LIN {X 0,Y 442.361,Z 632.864,A -85,B 0,C 180,E1 20654.481,E2 20654.481} C_VEL
LIN {X 0,Y 442.378,Z 633.008,A -85,B 0,C 180,E1 20653.963,E2 20653.963} C_VEL
LIN {X 0,Y 443.347,Z 635.847,A -85,B 0,C 180,E1 20653.617,E2 20653.617} C_VEL
LIN {X 0,Y 449.92,Z 650.433,A -85,B 0,C 180,E1 20651.693,E2 20651.693} C_VEL
LIN {X 0,Y 457.492,Z 669.791,A -85,B 0,C 180,E1 20649.312,E2 20649.312} C_VEL
LIN {X 0,Y 464.291,Z 690.305,A -85,B 0,C 180,E1 20646.967,E2 20646.967} C_VEL
LIN {X 0,Y 466.418,Z 698.2,A -85,B 0,C 180,E1 20646.121,E2 20646.121} C_VEL
LIN {X 0,Y 463.345,Z 744.603,A -85,B 0,C 180,E1 20642.434,E2 20642.434} C_VEL
LIN {X 0,Y 460.284,Z 791.954,A -85,B 0,C 180,E1 20638.689,E2 20638.689} C_VEL
LIN {X 0,Y 457.632,Z 840.214,A -85,B 0,C 180,E1 20634.996,E2 20634.996} C_VEL
LIN {X 0,Y 456.966,Z 857.735,A -85,B 0,C 180,E1 20633.736,E2 20633.736} C_VEL
LIN {X 0,Y 457.546,Z 865.068,A -85,B 0,C 180,E1 20633.578,E2 20633.578} C_VEL
LIN {X 0,Y 454.351,Z 1025.223,A -85,B 0,C 180,E1 20631.032,E2 20631.032} C_VEL
LIN {X 0,Y 453.962,Z 1043.295,A -85,B 0,C 180,E1 20630.535,E2 20630.535} C_VEL
LIN {X 0,Y 453.251,Z 1059.664,A -85,B 0,C 180,E1 20629.858,E2 20629.858} C_VEL
LIN {X 0,Y 452.212,Z 1075.509,A -85,B 0,C 180,E1 20628.965,E2 20628.965} C_VEL
LIN {X 0,Y 450.872,Z 1091.243,A -85,B 0,C 180,E1 20627.819,E2 20627.819} C_VEL
LIN {X 0,Y 449.462,Z 1105.194,A -85,B 0,C 180,E1 20626.542,E2 20626.542} C_VEL
LIN {X 0,Y 447.963,Z 1118.231,A -85,B 0,C 180,E1 20625.07,E2 20625.07} C_VEL
LIN {X 0,Y 446.506,Z 1129.751,A -85,B 0,C 180,E1 20623.465,E2 20623.465} C_VEL
LIN {X 0,Y 445.09,Z 1140.448,A -85,B 0,C 180,E1 20621.628,E2 20621.628} C_VEL
LIN {X 0,Y 443.836,Z 1149.901,A -85,B 0,C 180,E1 20619.595,E2 20619.595} C_VEL
LIN {X 0,Y 442.873,Z 1157.352,A -85,B 0,C 180,E1 20617.523,E2 20617.523} C_VEL
LIN {X 0,Y 442.159,Z 1163.241,A -85,B 0,C 180,E1 20615.318,E2 20615.318} C_VEL
LIN {X 0,Y 441.708,Z 1167.308,A -85,B 0,C 180,E1 20613.113,E2 20613.113} C_VEL
LIN {X 0,Y 441.474,Z 1169.774,A -85,B 0,C 180,E1 20610.777,E2 20610.777} C_VEL
LIN {X 0,Y 441.429,Z 1170.363,A -85,B 0,C 180,E1 20608.441,E2 20608.441} C_VEL
LIN {X 0,Y 441.579,Z 1169.177,A -85,B 0,C 180,E1 20606.103,E2 20606.103} C_VEL
LIN {X 0,Y 441.927,Z 1166.376,A -85,B 0,C 180,E1 20603.894,E2 20603.894} C_VEL
LIN {X 0,Y 442.053,Z 1165.325,A -85,B 0,C 180,E1 20603.317,E2 20603.317} C_VEL
LIN {X 0,Y 441.321,Z 1163.494,A -85,B 0,C 180,E1 20602.344,E2 20602.344} C_VEL
LIN {X 0,Y 436.574,Z 1158.567,A -85,B 0,C 180,E1 20600.104,E2 20600.104} C_VEL
LIN {X 0,Y 435.691,Z 1155.543,A -85,B 0,C 180,E1 20599.088,E2 20599.088} C_VEL
LIN {X 0,Y 435.74,Z 1155.097,A -85,B 0,C 180,E1 20598.953,E2 20598.953} C_VEL
LIN {X 0,Y 436.956,Z 1146.938,A -85,B 0,C 180,E1 20596.905,E2 20596.905} C_VEL
LIN {X 0,Y 438.441,Z 1136.934,A -85,B 0,C 180,E1 20594.929,E2 20594.929} C_VEL
LIN {X 0,Y 439.985,Z 1126.234,A -85,B 0,C 180,E1 20593.223,E2 20593.223} C_VEL
LIN {X 0,Y 441.676,Z 1113.643,A -85,B 0,C 180,E1 20591.589,E2 20591.589} C_VEL
LIN {X 0,Y 443.34,Z 1099.655,A -85,B 0,C 180,E1 20590.134,E2 20590.134} C_VEL
LIN {X 0,Y 444.89,Z 1084.381,A -85,B 0,C 180,E1 20588.863,E2 20588.863} C_VEL
LIN {X 0,Y 446.207,Z 1068.28,A -85,B 0,C 180,E1 20587.814,E2 20587.814} C_VEL
LIN {X 0,Y 447.186,Z 1051.309,A -85,B 0,C 180,E1 20586.994,E2 20586.994} C_VEL
LIN {X 0,Y 447.792,Z 1033.412,A -85,B 0,C 180,E1 20586.391,E2 20586.391} C_VEL
LIN {X 0,Y 448.019,Z 1011.916,A -85,B 0,C 180,E1 20585.965,E2 20585.965} C_VEL
LIN {X 0,Y 451.206,Z 862.917,A -85,B 0,C 180,E1 20583.572,E2 20583.572} C_VEL
LIN {X 0,Y 450.631,Z 858.057,A -85,B 0,C 180,E1 20583.441,E2 20583.441} C_VEL
LIN {X 0,Y 453.107,Z 811.957,A -85,B 0,C 180,E1 20579.937,E2 20579.937} C_VEL
LIN {X 0,Y 456.239,Z 765.453,A -85,B 0,C 180,E1 20576.249,E2 20576.249} C_VEL
LIN {X 0,Y 459.516,Z 719.315,A -85,B 0,C 180,E1 20572.548,E2 20572.548} C_VEL
LIN {X 0,Y 460.586,Z 701.904,A -85,B 0,C 180,E1 20571.141,E2 20571.141} C_VEL
LIN {X 0,Y 454.384,Z 682.18,A -85,B 0,C 180,E1 20568.854,E2 20568.854} C_VEL
LIN {X 0,Y 452.123,Z 675.599,A -85,B 0,C 180,E1 20568.03,E2 20568.03} C_VEL
LIN {X 0,Y 453.874,Z 676.346,A -85,B 0,C 180,E1 20567.783,E2 20567.783} C_VEL
LIN {X 0,Y 456.65,Z 675.663,A -85,B 0,C 180,E1 20567.463,E2 20567.463} C_VEL
LIN {X 0,Y 457.757,Z 675.439,A -85,B 0,C 180,E1 20567.335,E2 20567.335} C_VEL
LIN {X 0,Y 475.007,Z 699.868,A -85,B 0,C 180,E1 20564.535,E2 20564.535} C_VEL
LIN {X 0,Y 489.761,Z 721.8,A -85,B 0,C 180,E1 20562.337,E2 20562.337} C_VEL
LIN {X 0,Y 471.768,Z 976.974,A -85,B 0,C 180,E1 20557.054,E2 20557.054} C_VEL
LIN {X 0,Y 469.932,Z 1000.353,A -85,B 0,C 180,E1 20556.346,E2 20556.346} C_VEL
LIN {X 0,Y 467.68,Z 1022.366,A -85,B 0,C 180,E1 20555.476,E2 20555.476} C_VEL
LIN {X 0,Y 465.047,Z 1043.255,A -85,B 0,C 180,E1 20554.435,E2 20554.435} C_VEL
LIN {X 0,Y 461.875,Z 1064.722,A -85,B 0,C 180,E1 20553.136,E2 20553.136} C_VEL
LIN {X 0,Y 458.629,Z 1084.634,A -85,B 0,C 180,E1 20551.697,E2 20551.697} C_VEL
LIN {X 0,Y 455.16,Z 1103.712,A -85,B 0,C 180,E1 20550.054,E2 20550.054} C_VEL
LIN {X 0,Y 451.494,Z 1122.574,A -85,B 0,C 180,E1 20548.146,E2 20548.146} C_VEL
LIN {X 0,Y 447.975,Z 1139.989,A -85,B 0,C 180,E1 20546.085,E2 20546.085} C_VEL
LIN {X 0,Y 444.684,Z 1155.904,A -85,B 0,C 180,E1 20543.875,E2 20543.875} C_VEL
LIN {X 0,Y 441.628,Z 1170.646,A -85,B 0,C 180,E1 20541.478,E2 20541.478} C_VEL
LIN {X 0,Y 439.042,Z 1183.69,A -85,B 0,C 180,E1 20539.007,E2 20539.007} C_VEL
LIN {X 0,Y 436.819,Z 1195.499,A -85,B 0,C 180,E1 20536.353,E2 20536.353} C_VEL
LIN {X 0,Y 435.035,Z 1205.998,A -85,B 0,C 180,E1 20533.53,E2 20533.53} C_VEL
LIN {X 0,Y 433.8,Z 1214.56,A -85,B 0,C 180,E1 20530.76,E2 20530.76} C_VEL
LIN {X 0,Y 432.983,Z 1221.42,A -85,B 0,C 180,E1 20527.964,E2 20527.964} C_VEL
LIN {X 0,Y 432.473,Z 1227.215,A -85,B 0,C 180,E1 20524.907,E2 20524.907} C_VEL
LIN {X 0,Y 432.262,Z 1231,A -85,B 0,C 180,E1 20522.121,E2 20522.121} C_VEL
LIN {X 0,Y 432.189,Z 1233.379,A -85,B 0,C 180,E1 20519.205,E2 20519.205} C_VEL
LIN {X 0,Y 432.208,Z 1234.345,A -85,B 0,C 180,E1 20516.419,E2 20516.419} C_VEL
LIN {X 0,Y 432.276,Z 1233.807,A -85,B 0,C 180,E1 20513.625,E2 20513.625} C_VEL
LIN {X 0,Y 432.492,Z 1231.87,A -85,B 0,C 180,E1 20510.687,E2 20510.687} C_VEL
LIN {X 0,Y 432.906,Z 1228.535,A -85,B 0,C 180,E1 20507.867,E2 20507.867} C_VEL
LIN {X 0,Y 433.692,Z 1223.483,A -85,B 0,C 180,E1 20504.899,E2 20504.899} C_VEL
LIN {X 0,Y 434.909,Z 1217.159,A -85,B 0,C 180,E1 20502.057,E2 20502.057} C_VEL
LIN {X 0,Y 436.66,Z 1209.045,A -85,B 0,C 180,E1 20499.211,E2 20499.211} C_VEL
LIN {X 0,Y 439.038,Z 1199.132,A -85,B 0,C 180,E1 20496.37,E2 20496.37} C_VEL
LIN {X 0,Y 441.963,Z 1187.801,A -85,B 0,C 180,E1 20493.677,E2 20493.677} C_VEL
LIN {X 0,Y 445.374,Z 1174.918,A -85,B 0,C 180,E1 20491.115,E2 20491.115} C_VEL
LIN {X 0,Y 449.088,Z 1160.665,A -85,B 0,C 180,E1 20488.75,E2 20488.75} C_VEL
LIN {X 0,Y 452.879,Z 1145.755,A -85,B 0,C 180,E1 20486.65,E2 20486.65} C_VEL
LIN {X 0,Y 456.84,Z 1129.478,A -85,B 0,C 180,E1 20484.702,E2 20484.702} C_VEL
LIN {X 0,Y 460.685,Z 1112.341,A -85,B 0,C 180,E1 20482.965,E2 20482.965} C_VEL
LIN {X 0,Y 464.478,Z 1093.552,A -85,B 0,C 180,E1 20481.37,E2 20481.37} C_VEL
LIN {X 0,Y 467.935,Z 1073.587,A -85,B 0,C 180,E1 20479.97,E2 20479.97} C_VEL
LIN {X 0,Y 471.001,Z 1052.378,A -85,B 0,C 180,E1 20478.764,E2 20478.764} C_VEL
LIN {X 0,Y 473.486,Z 1030.442,A -85,B 0,C 180,E1 20477.783,E2 20477.783} C_VEL
LIN {X 0,Y 475.36,Z 1007.879,A -85,B 0,C 180,E1 20477.012,E2 20477.012} C_VEL
LIN {X 0,Y 478.712,Z 978.56,A -85,B 0,C 180,E1 20476.153,E2 20476.153} C_VEL
LIN {X 0,Y 484.513,Z 946.475,A -85,B 0,C 180,E1 20475.242,E2 20475.242} C_VEL
LIN {X 0,Y 493.348,Z 909.949,A -85,B 0,C 180,E1 20474.196,E2 20474.196} C_VEL
LIN {X 0,Y 491.563,Z 920.862,A -85,B 0,C 180,E1 20472.901,E2 20472.901} C_VEL
LIN {X 0,Y 491.452,Z 927.421,A -85,B 0,C 180,E1 20472.156,E2 20472.156} C_VEL
LIN {X 0,Y 485.87,Z 946.673,A -85,B 0,C 180,E1 20472.006,E2 20472.006} C_VEL
LIN {X 0,Y 480.627,Z 965.886,A -85,B 0,C 180,E1 20471.62,E2 20471.62} C_VEL
LIN {X 0,Y 476.101,Z 984.154,A -85,B 0,C 180,E1 20471.02,E2 20471.02} C_VEL
LIN {X 0,Y 467.969,Z 1021.759,A -85,B 0,C 180,E1 20469.32,E2 20469.32} C_VEL
LIN {X 0,Y 461.485,Z 1054.214,A -85,B 0,C 180,E1 20467.585,E2 20467.585} C_VEL
LIN {X 0,Y 455.667,Z 1086.671,A -85,B 0,C 180,E1 20465.558,E2 20465.558} C_VEL
LIN {X 0,Y 450.935,Z 1115.987,A -85,B 0,C 180,E1 20463.438,E2 20463.438} C_VEL
LIN {X 0,Y 446.734,Z 1144.254,A -85,B 0,C 180,E1 20461.086,E2 20461.086} C_VEL
LIN {X 0,Y 443.422,Z 1168.395,A -85,B 0,C 180,E1 20458.78,E2 20458.78} C_VEL
LIN {X 0,Y 440.588,Z 1189.873,A -85,B 0,C 180,E1 20456.413,E2 20456.413} C_VEL
LIN {X 0,Y 438.235,Z 1209.061,A -85,B 0,C 180,E1 20453.964,E2 20453.964} C_VEL
LIN {X 0,Y 436.417,Z 1224.669,A -85,B 0,C 180,E1 20451.648,E2 20451.648} C_VEL
LIN {X 0,Y 434.936,Z 1238.794,A -85,B 0,C 180,E1 20449.194,E2 20449.194} C_VEL
LIN {X 0,Y 433.801,Z 1250.64,A -85,B 0,C 180,E1 20446.747,E2 20446.747} C_VEL
LIN {X 0,Y 433.012,Z 1260.497,A -85,B 0,C 180,E1 20444.306,E2 20444.306} C_VEL
LIN {X 0,Y 432.506,Z 1268.942,A -85,B 0,C 180,E1 20441.74,E2 20441.74} C_VEL
LIN {X 0,Y 432.226,Z 1275.553,A -85,B 0,C 180,E1 20439.187,E2 20439.187} C_VEL
LIN {X 0,Y 432.141,Z 1280.686,A -85,B 0,C 180,E1 20436.512,E2 20436.512} C_VEL
LIN {X 0,Y 432.145,Z 1283.861,A -85,B 0,C 180,E1 20433.982,E2 20433.982} C_VEL
LIN {X 0,Y 432.171,Z 1285.546,A -85,B 0,C 180,E1 20431.328,E2 20431.328} C_VEL
LIN {X 0,Y 432.169,Z 1285.595,A -85,B 0,C 180,E1 20428.676,E2 20428.676} C_VEL
LIN {X 0,Y 432.137,Z 1284.048,A -85,B 0,C 180,E1 20426.021,E2 20426.021} C_VEL
LIN {X 0,Y 432.118,Z 1280.876,A -85,B 0,C 180,E1 20423.358,E2 20423.358} C_VEL
LIN {X 0,Y 432.221,Z 1275.811,A -85,B 0,C 180,E1 20420.548,E2 20420.548} C_VEL
LIN {X 0,Y 432.552,Z 1268.98,A -85,B 0,C 180,E1 20417.723,E2 20417.723} C_VEL
LIN {X 0,Y 433.259,Z 1259.669,A -85,B 0,C 180,E1 20414.726,E2 20414.726} C_VEL
LIN {X 0,Y 434.381,Z 1248.907,A -85,B 0,C 180,E1 20411.898,E2 20411.898} C_VEL
LIN {X 0,Y 436.057,Z 1235.907,A -85,B 0,C 180,E1 20409.042,E2 20409.042} C_VEL
LIN {X 0,Y 438.251,Z 1221.293,A -85,B 0,C 180,E1 20406.327,E2 20406.327} C_VEL
LIN {X 0,Y 440.94,Z 1205.226,A -85,B 0,C 180,E1 20403.759,E2 20403.759} C_VEL
LIN {X 0,Y 444.345,Z 1186.33,A -85,B 0,C 180,E1 20401.163,E2 20401.163} C_VEL
LIN {X 0,Y 448.432,Z 1164.856,A -85,B 0,C 180,E1 20398.649,E2 20398.649} C_VEL
LIN {X 0,Y 452.655,Z 1143.094,A -85,B 0,C 180,E1 20396.482,E2 20396.482} C_VEL
LIN {X 0,Y 457.071,Z 1120.987,A -85,B 0,C 180,E1 20394.572,E2 20394.572} C_VEL
LIN {X 0,Y 461.561,Z 1097.922,A -85,B 0,C 180,E1 20392.887,E2 20392.887} C_VEL
LIN {X 0,Y 466.241,Z 1073.881,A -85,B 0,C 180,E1 20391.389,E2 20391.389} C_VEL
LIN {X 0,Y 470.405,Z 1051.347,A -85,B 0,C 180,E1 20390.226,E2 20390.226} C_VEL
LIN {X 0,Y 474.759,Z 1026.579,A -85,B 0,C 180,E1 20389.163,E2 20389.163} C_VEL
LIN {X 0,Y 478.579,Z 1001.615,A -85,B 0,C 180,E1 20388.317,E2 20388.317} C_VEL
LIN {X 0,Y 481.845,Z 975.438,A -85,B 0,C 180,E1 20387.621,E2 20387.621} C_VEL
LIN {X 0,Y 485.239,Z 953.953,A -85,B 0,C 180,E1 20387.28,E2 20387.28} C_VEL
LIN {X 0,Y 485.44,Z 951.656,A -85,B 0,C 180,E1 20387.232,E2 20387.232} C_VEL
LIN {X 0,Y 475.455,Z 930.968,A -85,B 0,C 180,E1 20385.71,E2 20385.71} C_VEL
LIN {X 0,Y 473.644,Z 926.121,A -85,B 0,C 180,E1 20385.351,E2 20385.351} C_VEL
LIN {X 0,Y 470.533,Z 906.683,A -85,B 0,C 180,E1 20383.011,E2 20383.011} C_VEL
LIN {X 0,Y 469.842,Z 885.654,A -85,B 0,C 180,E1 20380.633,E2 20380.633} C_VEL
LIN {X 0,Y 471.699,Z 862.2,A -85,B 0,C 180,E1 20378.15,E2 20378.15} C_VEL
LIN {X 0,Y 478.112,Z 821.82,A -85,B 0,C 180,E1 20374.089,E2 20374.089} C_VEL
LIN {X 0,Y 483.755,Z 787.898,A -85,B 0,C 180,E1 20370.638,E2 20370.638} C_VEL
LIN {X 0,Y 489.081,Z 756.617,A -85,B 0,C 180,E1 20367.387,E2 20367.387} C_VEL
LIN {X 0,Y 482.488,Z 739.607,A -85,B 0,C 180,E1 20364.356,E2 20364.356} C_VEL
LIN {X 0,Y 475.807,Z 723.064,A -85,B 0,C 180,E1 20361.189,E2 20361.189} C_VEL
LIN {X 0,Y 468.783,Z 706.507,A -85,B 0,C 180,E1 20357.759,E2 20357.759} C_VEL
LIN {X 0,Y 461.708,Z 690.572,A -85,B 0,C 180,E1 20354.165,E2 20354.165} C_VEL
LIN {X 0,Y 455.438,Z 677.174,A -85,B 0,C 180,E1 20350.883,E2 20350.883} C_VEL
LIN {X 0,Y 449.891,Z 665.361,A -85,B 0,C 180,E1 20347.792,E2 20347.792} C_VEL
LIN {X 0,Y 445.031,Z 655.663,A -85,B 0,C 180,E1 20345.027,E2 20345.027} C_VEL
LIN {X 0,Y 442.88,Z 651.358,A -85,B 0,C 180,E1 20343.75,E2 20343.75} C_VEL
LIN {X 0,Y 440.804,Z 647.144,A -85,B 0,C 180,E1 20342.47,E2 20342.47} C_VEL
LIN {X 0,Y 438.787,Z 642.92,A -85,B 0,C 180,E1 20341.175,E2 20341.175} C_VEL
LIN {X 0,Y 436.932,Z 639.254,A -85,B 0,C 180,E1 20339.98,E2 20339.98} C_VEL
LIN {X 0,Y 434.526,Z 634.515,A -85,B 0,C 180,E1 20338.418,E2 20338.418} C_VEL
LIN {X 0,Y 434.411,Z 633.857,A -85,B 0,C 180,E1 20338.153,E2 20338.153} C_VEL
LIN {X 0,Y 434.42,Z 633.869,A -85,B 0,C 180,E1 20334.32,E2 20334.32} C_VEL
LIN {X 0,Y 434.41,Z 633.863,A -85,B 0,C 180,E1 20330.594,E2 20330.594} C_VEL
LIN {X 0,Y 434.421,Z 633.855,A -85,B 0,C 180,E1 20326.693,E2 20326.693} C_VEL
LIN {X 0,Y 434.416,Z 633.857,A -85,B 0,C 180,E1 20323.003,E2 20323.003} C_VEL
LIN {X 0,Y 434.41,Z 633.861,A -85,B 0,C 180,E1 20319.239,E2 20319.239} C_VEL
LIN {X 0,Y 434.422,Z 633.863,A -85,B 0,C 180,E1 20315.38,E2 20315.38} C_VEL
LIN {X 0,Y 434.425,Z 633.863,A -85,B 0,C 180,E1 20311.544,E2 20311.544} C_VEL
LIN {X 0,Y 434.412,Z 633.866,A -85,B 0,C 180,E1 20307.724,E2 20307.724} C_VEL
LIN {X 0,Y 434.415,Z 633.859,A -85,B 0,C 180,E1 20304.06,E2 20304.06} C_VEL
LIN {X 0,Y 434.424,Z 633.863,A -85,B 0,C 180,E1 20300.219,E2 20300.219} C_VEL
LIN {X 0,Y 434.41,Z 633.817,A -85,B 0,C 180,E1 20296.329,E2 20296.329} C_VEL
LIN {X 0,Y 434.418,Z 633.853,A -85,B 0,C 180,E1 20294.771,E2 20294.771} C_VEL
LIN {X 0,Y 435.357,Z 636.731,A -85,B 0,C 180,E1 20294.416,E2 20294.416} C_VEL
LIN {X 0,Y 439.742,Z 646.024,A -85,B 0,C 180,E1 20293.122,E2 20293.122} C_VEL
LIN {X 0,Y 447.436,Z 664.476,A -85,B 0,C 180,E1 20290.73,E2 20290.73} C_VEL
LIN {X 0,Y 454.706,Z 684.886,A -85,B 0,C 180,E1 20288.275,E2 20288.275} C_VEL
LIN {X 0,Y 459.428,Z 700.781,A -85,B 0,C 180,E1 20286.5,E2 20286.5} C_VEL
LIN {X 0,Y 456.328,Z 745.479,A -85,B 0,C 180,E1 20282.913,E2 20282.913} C_VEL
LIN {X 0,Y 453.203,Z 792.434,A -85,B 0,C 180,E1 20279.18,E2 20279.18} C_VEL
LIN {X 0,Y 450.475,Z 840.077,A -85,B 0,C 180,E1 20275.504,E2 20275.504} C_VEL
LIN {X 0,Y 449.716,Z 858.67,A -85,B 0,C 180,E1 20274.153,E2 20274.153} C_VEL
LIN {X 0,Y 450.277,Z 866.044,A -85,B 0,C 180,E1 20273.992,E2 20273.992} C_VEL
LIN {X 0,Y 446.961,Z 1025.867,A -85,B 0,C 180,E1 20271.414,E2 20271.414} C_VEL
LIN {X 0,Y 446.556,Z 1044.024,A -85,B 0,C 180,E1 20270.909,E2 20270.909} C_VEL
LIN {X 0,Y 445.799,Z 1060.815,A -85,B 0,C 180,E1 20270.205,E2 20270.205} C_VEL
LIN {X 0,Y 444.719,Z 1076.607,A -85,B 0,C 180,E1 20269.298,E2 20269.298} C_VEL
LIN {X 0,Y 443.33,Z 1092.314,A -85,B 0,C 180,E1 20268.132,E2 20268.132} C_VEL
LIN {X 0,Y 441.843,Z 1106.464,A -85,B 0,C 180,E1 20266.813,E2 20266.813} C_VEL
LIN {X 0,Y 440.24,Z 1119.753,A -85,B 0,C 180,E1 20265.274,E2 20265.274} C_VEL
LIN {X 0,Y 438.68,Z 1131.583,A -85,B 0,C 180,E1 20263.576,E2 20263.576} C_VEL
LIN {X 0,Y 437.25,Z 1141.953,A -85,B 0,C 180,E1 20261.741,E2 20261.741} C_VEL
LIN {X 0,Y 436.009,Z 1150.899,A -85,B 0,C 180,E1 20259.769,E2 20259.769} C_VEL
LIN {X 0,Y 435,Z 1158.338,A -85,B 0,C 180,E1 20257.659,E2 20257.659} C_VEL
LIN {X 0,Y 434.252,Z 1164.219,A -85,B 0,C 180,E1 20255.415,E2 20255.415} C_VEL
LIN {X 0,Y 433.778,Z 1168.278,A -85,B 0,C 180,E1 20253.169,E2 20253.169} C_VEL
LIN {X 0,Y 433.533,Z 1170.732,A -85,B 0,C 180,E1 20250.791,E2 20250.791} C_VEL
LIN {X 0,Y 433.486,Z 1171.314,A -85,B 0,C 180,E1 20248.412,E2 20248.412} C_VEL
LIN {X 0,Y 433.647,Z 1170.121,A -85,B 0,C 180,E1 20246.032,E2 20246.032} C_VEL
LIN {X 0,Y 434.017,Z 1167.313,A -85,B 0,C 180,E1 20243.782,E2 20243.782} C_VEL
LIN {X 0,Y 434.642,Z 1162.71,A -85,B 0,C 180,E1 20241.532,E2 20241.532} C_VEL
LIN {X 0,Y 435.576,Z 1156.142,A -85,B 0,C 180,E1 20239.267,E2 20239.267} C_VEL
LIN {X 0,Y 435.74,Z 1155.097,A -85,B 0,C 180,E1 20238.953,E2 20238.953} C_VEL
LIN {X 0,Y 435.289,Z 1151.958,A -85,B 0,C 180,E1 20238.02,E2 20238.02} C_VEL
LIN {X 0,Y 431.73,Z 1145.302,A -85,B 0,C 180,E1 20236.204,E2 20236.204} C_VEL
LIN {X 0,Y 430.511,Z 1140.757,A -85,B 0,C 180,E1 20235.199,E2 20235.199} C_VEL
LIN {X 0,Y 430.603,Z 1138.835,A -85,B 0,C 180,E1 20234.836,E2 20234.836} C_VEL
LIN {X 0,Y 432.368,Z 1127.107,A -85,B 0,C 180,E1 20232.919,E2 20232.919} C_VEL
LIN {X 0,Y 434.13,Z 1114.495,A -85,B 0,C 180,E1 20231.257,E2 20231.257} C_VEL
LIN {X 0,Y 435.836,Z 1100.708,A -85,B 0,C 180,E1 20229.8,E2 20229.8} C_VEL
LIN {X 0,Y 437.397,Z 1085.929,A -85,B 0,C 180,E1 20228.544,E2 20228.544} C_VEL
LIN {X 0,Y 438.753,Z 1070.125,A -85,B 0,C 180,E1 20227.487,E2 20227.487} C_VEL
LIN {X 0,Y 439.79,Z 1053.487,A -85,B 0,C 180,E1 20226.651,E2 20226.651} C_VEL
LIN {X 0,Y 440.432,Z 1035.997,A -85,B 0,C 180,E1 20226.035,E2 20226.035} C_VEL
LIN {X 0,Y 440.682,Z 1016.129,A -85,B 0,C 180,E1 20225.61,E2 20225.61} C_VEL
LIN {X 0,Y 444.041,Z 863.864,A -85,B 0,C 180,E1 20223.126,E2 20223.126} C_VEL
LIN {X 0,Y 443.473,Z 859.061,A -85,B 0,C 180,E1 20222.995,E2 20222.995} C_VEL
LIN {X 0,Y 445.981,Z 814.116,A -85,B 0,C 180,E1 20219.555,E2 20219.555} C_VEL
LIN {X 0,Y 449.23,Z 767.039,A -85,B 0,C 180,E1 20215.804,E2 20215.804} C_VEL
LIN {X 0,Y 452.602,Z 721.3,A -85,B 0,C 180,E1 20212.108,E2 20212.108} C_VEL
LIN {X 0,Y 453.655,Z 704.806,A -85,B 0,C 180,E1 20210.758,E2 20210.758} C_VEL
LIN {X 0,Y 447.346,Z 684.549,A -85,B 0,C 180,E1 20208.341,E2 20208.341} C_VEL
LIN {X 0,Y 449.089,Z 685.28,A -85,B 0,C 180,E1 20208.09,E2 20208.09} C_VEL
LIN {X 0,Y 451.836,Z 684.583,A -85,B 0,C 180,E1 20207.763,E2 20207.763} C_VEL
LIN {X 0,Y 453.495,Z 684.211,A -85,B 0,C 180,E1 20207.569,E2 20207.569} C_VEL
LIN {X 0,Y 455.12,Z 684.122,A -85,B 0,C 180,E1 20207.372,E2 20207.372} C_VEL
LIN {X 0,Y 470.635,Z 706.14,A -85,B 0,C 180,E1 20204.839,E2 20204.839} C_VEL
LIN {X 0,Y 483.472,Z 725.409,A -85,B 0,C 180,E1 20202.882,E2 20202.882} C_VEL
LIN {X 0,Y 464.924,Z 977.284,A -85,B 0,C 180,E1 20197.559,E2 20197.559} C_VEL
LIN {X 0,Y 462.962,Z 1001.559,A -85,B 0,C 180,E1 20196.813,E2 20196.813} C_VEL
LIN {X 0,Y 460.532,Z 1024.321,A -85,B 0,C 180,E1 20195.889,E2 20195.889} C_VEL
LIN {X 0,Y 457.648,Z 1046.328,A -85,B 0,C 180,E1 20194.763,E2 20194.763} C_VEL
LIN {X 0,Y 454.42,Z 1067.268,A -85,B 0,C 180,E1 20193.449,E2 20193.449} C_VEL
LIN {X 0,Y 450.743,Z 1088.767,A -85,B 0,C 180,E1 20191.828,E2 20191.828} C_VEL
LIN {X 0,Y 447.189,Z 1107.79,A -85,B 0,C 180,E1 20190.131,E2 20190.131} C_VEL
LIN {X 0,Y 443.573,Z 1125.568,A -85,B 0,C 180,E1 20188.254,E2 20188.254} C_VEL
LIN {X 0,Y 439.805,Z 1143.593,A -85,B 0,C 180,E1 20186.026,E2 20186.026} C_VEL
LIN {X 0,Y 436.496,Z 1159.188,A -85,B 0,C 180,E1 20183.776,E2 20183.776} C_VEL
LIN {X 0,Y 433.492,Z 1173.353,A -85,B 0,C 180,E1 20181.373,E2 20181.373} C_VEL
LIN {X 0,Y 430.72,Z 1186.835,A -85,B 0,C 180,E1 20178.685,E2 20178.685} C_VEL
LIN {X 0,Y 428.554,Z 1198.321,A -85,B 0,C 180,E1 20175.981,E2 20175.981} C_VEL
LIN {X 0,Y 426.902,Z 1207.9,A -85,B 0,C 180,E1 20173.27,E2 20173.27} C_VEL
LIN {X 0,Y 425.64,Z 1216.58,A -85,B 0,C 180,E1 20170.285,E2 20170.285} C_VEL
LIN {X 0,Y 424.889,Z 1223.242,A -85,B 0,C 180,E1 20167.437,E2 20167.437} C_VEL
LIN {X 0,Y 424.452,Z 1228.23,A -85,B 0,C 180,E1 20164.594,E2 20164.594} C_VEL
LIN {X 0,Y 424.256,Z 1232.01,A -85,B 0,C 180,E1 20161.621,E2 20161.621} C_VEL
LIN {X 0,Y 424.204,Z 1234.09,A -85,B 0,C 180,E1 20158.784,E2 20158.784} C_VEL
LIN {X 0,Y 424.228,Z 1234.843,A -85,B 0,C 180,E1 20155.674,E2 20155.674} C_VEL
LIN {X 0,Y 424.359,Z 1234.079,A -85,B 0,C 180,E1 20152.745,E2 20152.745} C_VEL
LIN {X 0,Y 424.625,Z 1231.795,A -85,B 0,C 180,E1 20149.828,E2 20149.828} C_VEL
LIN {X 0,Y 425.204,Z 1227.975,A -85,B 0,C 180,E1 20146.795,E2 20146.795} C_VEL
LIN {X 0,Y 426.19,Z 1222.575,A -85,B 0,C 180,E1 20143.788,E2 20143.788} C_VEL
LIN {X 0,Y 427.739,Z 1215.379,A -85,B 0,C 180,E1 20140.755,E2 20140.755} C_VEL
LIN {X 0,Y 429.958,Z 1206.349,A -85,B 0,C 180,E1 20137.724,E2 20137.724} C_VEL
LIN {X 0,Y 432.665,Z 1196.259,A -85,B 0,C 180,E1 20134.949,E2 20134.949} C_VEL
LIN {X 0,Y 435.967,Z 1184.372,A -85,B 0,C 180,E1 20132.252,E2 20132.252} C_VEL
LIN {X 0,Y 439.559,Z 1171.576,A -85,B 0,C 180,E1 20129.817,E2 20129.817} C_VEL
LIN {X 0,Y 443.724,Z 1156.639,A -85,B 0,C 180,E1 20127.414,E2 20127.414} C_VEL
LIN {X 0,Y 447.913,Z 1141.065,A -85,B 0,C 180,E1 20125.302,E2 20125.302} C_VEL
LIN {X 0,Y 452.078,Z 1124.597,A -85,B 0,C 180,E1 20123.407,E2 20123.407} C_VEL
LIN {X 0,Y 456.398,Z 1105.826,A -85,B 0,C 180,E1 20121.603,E2 20121.603} C_VEL
LIN {X 0,Y 460.354,Z 1086.475,A -85,B 0,C 180,E1 20120.062,E2 20120.062} C_VEL
LIN {X 0,Y 463.78,Z 1066.993,A -85,B 0,C 180,E1 20118.777,E2 20118.777} C_VEL
LIN {X 0,Y 466.898,Z 1045.987,A -85,B 0,C 180,E1 20117.652,E2 20117.652} C_VEL
LIN {X 0,Y 469.446,Z 1024.223,A -85,B 0,C 180,E1 20116.733,E2 20116.733} C_VEL
LIN {X 0,Y 472.881,Z 994.654,A -85,B 0,C 180,E1 20115.751,E2 20115.751} C_VEL
LIN {X 0,Y 478.194,Z 966.7,A -85,B 0,C 180,E1 20114.891,E2 20114.891} C_VEL
LIN {X 0,Y 486.634,Z 934.282,A -85,B 0,C 180,E1 20113.931,E2 20113.931} C_VEL
LIN {X 0,Y 489.317,Z 925.284,A -85,B 0,C 180,E1 20113.649,E2 20113.649} C_VEL
LIN {X 0,Y 488.556,Z 930.278,A -85,B 0,C 180,E1 20113.053,E2 20113.053} C_VEL
LIN {X 0,Y 482.971,Z 949.556,A -85,B 0,C 180,E1 20112.878,E2 20112.878} C_VEL
LIN {X 0,Y 477.573,Z 968.489,A -85,B 0,C 180,E1 20112.472,E2 20112.472} C_VEL
LIN {X 0,Y 472.734,Z 986.225,A -85,B 0,C 180,E1 20111.862,E2 20111.862} C_VEL
LIN {X 0,Y 463.443,Z 1023.785,A -85,B 0,C 180,E1 20110.094,E2 20110.094} C_VEL
LIN {X 0,Y 456.064,Z 1056.427,A -85,B 0,C 180,E1 20108.271,E2 20108.271} C_VEL
LIN {X 0,Y 449.291,Z 1090.143,A -85,B 0,C 180,E1 20106.062,E2 20106.062} C_VEL
LIN {X 0,Y 443.848,Z 1120.553,A -85,B 0,C 180,E1 20103.741,E2 20103.741} C_VEL
LIN {X 0,Y 439.027,Z 1150.054,A -85,B 0,C 180,E1 20101.132,E2 20101.132} C_VEL
LIN {X 0,Y 435.44,Z 1174.145,A -85,B 0,C 180,E1 20098.682,E2 20098.682} C_VEL
LIN {X 0,Y 432.481,Z 1195.161,A -85,B 0,C 180,E1 20096.207,E2 20096.207} C_VEL
LIN {X 0,Y 430.083,Z 1213.424,A -85,B 0,C 180,E1 20093.718,E2 20093.718} C_VEL
LIN {X 0,Y 428.165,Z 1229.129,A -85,B 0,C 180,E1 20091.223,E2 20091.223} C_VEL
LIN {X 0,Y 426.696,Z 1242.474,A -85,B 0,C 180,E1 20088.727,E2 20088.727} C_VEL
LIN {X 0,Y 425.619,Z 1253.67,A -85,B 0,C 180,E1 20086.236,E2 20086.236} C_VEL
LIN {X 0,Y 424.842,Z 1263.46,A -85,B 0,C 180,E1 20083.585,E2 20083.585} C_VEL
LIN {X 0,Y 424.386,Z 1271.478,A -85,B 0,C 180,E1 20080.866,E2 20080.866} C_VEL
LIN {X 0,Y 424.181,Z 1277.626,A -85,B 0,C 180,E1 20078.133,E2 20078.133} C_VEL
LIN {X 0,Y 424.143,Z 1281.751,A -85,B 0,C 180,E1 20075.548,E2 20075.548} C_VEL
LIN {X 0,Y 424.17,Z 1284.335,A -85,B 0,C 180,E1 20072.839,E2 20072.839} C_VEL
LIN {X 0,Y 424.202,Z 1285.246,A -85,B 0,C 180,E1 20070.137,E2 20070.137} C_VEL
LIN {X 0,Y 424.171,Z 1284.523,A -85,B 0,C 180,E1 20067.435,E2 20067.435} C_VEL
LIN {X 0,Y 424.145,Z 1282.193,A -85,B 0,C 180,E1 20064.727,E2 20064.727} C_VEL
LIN {X 0,Y 424.165,Z 1277.956,A -85,B 0,C 180,E1 20061.871,E2 20061.871} C_VEL
LIN {X 0,Y 424.371,Z 1271.96,A -85,B 0,C 180,E1 20059,E2 20059} C_VEL
LIN {X 0,Y 424.835,Z 1264.508,A -85,B 0,C 180,E1 20056.251,E2 20056.251} C_VEL
LIN {X 0,Y 425.726,Z 1254.78,A -85,B 0,C 180,E1 20053.351,E2 20053.351} C_VEL
LIN {X 0,Y 427.062,Z 1243.588,A -85,B 0,C 180,E1 20050.584,E2 20050.584} C_VEL
LIN {X 0,Y 429.04,Z 1229.649,A -85,B 0,C 180,E1 20047.676,E2 20047.676} C_VEL
LIN {X 0,Y 431.573,Z 1214.037,A -85,B 0,C 180,E1 20044.916,E2 20044.916} C_VEL
LIN {X 0,Y 434.629,Z 1196.884,A -85,B 0,C 180,E1 20042.311,E2 20042.311} C_VEL
LIN {X 0,Y 438.417,Z 1177.142,A -85,B 0,C 180,E1 20039.736,E2 20039.736} C_VEL
LIN {X 0,Y 442.695,Z 1155.617,A -85,B 0,C 180,E1 20037.332,E2 20037.332} C_VEL
LIN {X 0,Y 447.58,Z 1131.425,A -85,B 0,C 180,E1 20035.042,E2 20035.042} C_VEL
LIN {X 0,Y 451.931,Z 1110.129,A -85,B 0,C 180,E1 20033.321,E2 20033.321} C_VEL
LIN {X 0,Y 456.996,Z 1084.983,A -85,B 0,C 180,E1 20031.586,E2 20031.586} C_VEL
LIN {X 0,Y 461.453,Z 1062.22,A -85,B 0,C 180,E1 20030.27,E2 20030.27} C_VEL
LIN {X 0,Y 466.29,Z 1036.214,A -85,B 0,C 180,E1 20029.035,E2 20029.035} C_VEL
LIN {X 0,Y 470.607,Z 1011.13,A -85,B 0,C 180,E1 20028.074,E2 20028.074} C_VEL
LIN {X 0,Y 474.137,Z 985.021,A -85,B 0,C 180,E1 20027.285,E2 20027.285} C_VEL
LIN {X 0,Y 476.92,Z 965.187,A -85,B 0,C 180,E1 20026.861,E2 20026.861} C_VEL
LIN {X 0,Y 478.68,Z 954.162,A -85,B 0,C 180,E1 20026.694,E2 20026.694} C_VEL
LIN {X 0,Y 469.464,Z 934.685,A -85,B 0,C 180,E1 20025.238,E2 20025.238} C_VEL
LIN {X 0,Y 465.374,Z 923.825,A -85,B 0,C 180,E1 20024.462,E2 20024.462} C_VEL
LIN {X 0,Y 462.989,Z 904.169,A -85,B 0,C 180,E1 20022.111,E2 20022.111} C_VEL
LIN {X 0,Y 463.032,Z 882.287,A -85,B 0,C 180,E1 20019.644,E2 20019.644} C_VEL
LIN {X 0,Y 465.656,Z 858.172,A -85,B 0,C 180,E1 20017.113,E2 20017.113} C_VEL
LIN {X 0,Y 471.492,Z 823.054,A -85,B 0,C 180,E1 20013.551,E2 20013.551} C_VEL
LIN {X 0,Y 477.402,Z 788.954,A -85,B 0,C 180,E1 20010.038,E2 20010.038} C_VEL
LIN {X 0,Y 482.411,Z 760.261,A -85,B 0,C 180,E1 20007.029,E2 20007.029} C_VEL
LIN {X 0,Y 475.302,Z 741.849,A -85,B 0,C 180,E1 20003.691,E2 20003.691} C_VEL
LIN {X 0,Y 468.163,Z 724.265,A -85,B 0,C 180,E1 20000.243,E2 20000.243} C_VEL
LIN {X 0,Y 460.923,Z 707.32,A -85,B 0,C 180,E1 19996.64,E2 19996.64} C_VEL
LIN {X 0,Y 454.108,Z 692.108,A -85,B 0,C 180,E1 19993.108,E2 19993.108} C_VEL
LIN {X 0,Y 447.945,Z 678.865,A -85,B 0,C 180,E1 19989.767,E2 19989.767} C_VEL
LIN {X 0,Y 442.006,Z 666.375,A -85,B 0,C 180,E1 19986.364,E2 19986.364} C_VEL
LIN {X 0,Y 437.216,Z 656.814,A -85,B 0,C 180,E1 19983.54,E2 19983.54} C_VEL
LIN {X 0,Y 435.084,Z 652.559,A -85,B 0,C 180,E1 19982.239,E2 19982.239} C_VEL
LIN {X 0,Y 432.983,Z 648.255,A -85,B 0,C 180,E1 19980.881,E2 19980.881} C_VEL
LIN {X 0,Y 430.567,Z 643.531,A -85,B 0,C 180,E1 19979.335,E2 19979.335} C_VEL
LIN {X 0,Y 428.418,Z 639.162,A -85,B 0,C 180,E1 19977.86,E2 19977.86} C_VEL
LIN {X 0,Y 426.646,Z 635.8,A -85,B 0,C 180,E1 19976.686,E2 19976.686} C_VEL
LIN {X 0,Y 426.474,Z 634.85,A -85,B 0,C 180,E1 19976.371,E2 19976.371} C_VEL
LIN {X 0,Y 426.487,Z 634.844,A -85,B 0,C 180,E1 19972.456,E2 19972.456} C_VEL
LIN {X 0,Y 426.471,Z 634.856,A -85,B 0,C 180,E1 19968.505,E2 19968.505} C_VEL
LIN {X 0,Y 426.486,Z 634.856,A -85,B 0,C 180,E1 19964.637,E2 19964.637} C_VEL
LIN {X 0,Y 426.484,Z 634.849,A -85,B 0,C 180,E1 19960.696,E2 19960.696} C_VEL
LIN {X 0,Y 426.472,Z 634.847,A -85,B 0,C 180,E1 19956.949,E2 19956.949} C_VEL
LIN {X 0,Y 426.476,Z 634.843,A -85,B 0,C 180,E1 19953.246,E2 19953.246} C_VEL
LIN {X 0,Y 426.483,Z 634.842,A -85,B 0,C 180,E1 19949.419,E2 19949.419} C_VEL
LIN {X 0,Y 426.481,Z 634.841,A -85,B 0,C 180,E1 19945.596,E2 19945.596} C_VEL
LIN {X 0,Y 426.475,Z 634.844,A -85,B 0,C 180,E1 19941.756,E2 19941.756} C_VEL
LIN {X 0,Y 426.475,Z 634.821,A -85,B 0,C 180,E1 19938.003,E2 19938.003} C_VEL
LIN {X 0,Y 426.495,Z 634.974,A -85,B 0,C 180,E1 19935.588,E2 19935.588} C_VEL
LIN {X 0,Y 427.888,Z 638.468,A -85,B 0,C 180,E1 19935.112,E2 19935.112} C_VEL
LIN {X 0,Y 435.286,Z 654.729,A -85,B 0,C 180,E1 19932.836,E2 19932.836} C_VEL
LIN {X 0,Y 442.672,Z 673.219,A -85,B 0,C 180,E1 19930.429,E2 19930.429} C_VEL
LIN {X 0,Y 449.641,Z 693.771,A -85,B 0,C 180,E1 19927.981,E2 19927.981} C_VEL
LIN {X 0,Y 452.428,Z 703.626,A -85,B 0,C 180,E1 19926.866,E2 19926.866} C_VEL
LIN {X 0,Y 449.186,Z 749.091,A -85,B 0,C 180,E1 19923.2,E2 19923.2} C_VEL
LIN {X 0,Y 445.934,Z 796.449,A -85,B 0,C 180,E1 19919.407,E2 19919.407} C_VEL
LIN {X 0,Y 443.095,Z 844.611,A -85,B 0,C 180,E1 19915.673,E2 19915.673} C_VEL
LIN {X 0,Y 442.481,Z 859.519,A -85,B 0,C 180,E1 19914.586,E2 19914.586} C_VEL
LIN {X 0,Y 443.035,Z 866.897,A -85,B 0,C 180,E1 19914.421,E2 19914.421} C_VEL
LIN {X 0,Y 439.591,Z 1026.492,A -85,B 0,C 180,E1 19911.808,E2 19911.808} C_VEL
LIN {X 0,Y 439.173,Z 1044.654,A -85,B 0,C 180,E1 19911.3,E2 19911.3} C_VEL
LIN {X 0,Y 438.402,Z 1061.291,A -85,B 0,C 180,E1 19910.596,E2 19910.596} C_VEL
LIN {X 0,Y 437.326,Z 1076.74,A -85,B 0,C 180,E1 19909.707,E2 19909.707} C_VEL
LIN {X 0,Y 435.958,Z 1091.824,A -85,B 0,C 180,E1 19908.588,E2 19908.588} C_VEL
LIN {X 0,Y 434.423,Z 1106.012,A -85,B 0,C 180,E1 19907.27,E2 19907.27} C_VEL
LIN {X 0,Y 432.793,Z 1119.249,A -85,B 0,C 180,E1 19905.749,E2 19905.749} C_VEL
LIN {X 0,Y 431.206,Z 1130.971,A -85,B 0,C 180,E1 19904.09,E2 19904.09} C_VEL
LIN {X 0,Y 429.655,Z 1141.747,A -85,B 0,C 180,E1 19902.197,E2 19902.197} C_VEL
LIN {X 0,Y 428.26,Z 1151.345,A -85,B 0,C 180,E1 19900.083,E2 19900.083} C_VEL
LIN {X 0,Y 427.189,Z 1158.933,A -85,B 0,C 180,E1 19897.936,E2 19897.936} C_VEL
LIN {X 0,Y 426.385,Z 1164.905,A -85,B 0,C 180,E1 19895.65,E2 19895.65} C_VEL
LIN {X 0,Y 425.849,Z 1169.247,A -85,B 0,C 180,E1 19893.229,E2 19893.229} C_VEL
LIN {X 0,Y 425.591,Z 1171.69,A -85,B 0,C 180,E1 19890.806,E2 19890.806} C_VEL
LIN {X 0,Y 425.544,Z 1172.265,A -85,B 0,C 180,E1 19888.382,E2 19888.382} C_VEL
LIN {X 0,Y 425.716,Z 1171.065,A -85,B 0,C 180,E1 19885.958,E2 19885.958} C_VEL
LIN {X 0,Y 426.109,Z 1168.249,A -85,B 0,C 180,E1 19883.666,E2 19883.666} C_VEL
LIN {X 0,Y 426.768,Z 1163.635,A -85,B 0,C 180,E1 19881.374,E2 19881.374} C_VEL
LIN {X 0,Y 427.746,Z 1157.11,A -85,B 0,C 180,E1 19879.084,E2 19879.084} C_VEL
LIN {X 0,Y 429.02,Z 1149.015,A -85,B 0,C 180,E1 19876.932,E2 19876.932} C_VEL
LIN {X 0,Y 430.533,Z 1139.309,A -85,B 0,C 180,E1 19874.922,E2 19874.922} C_VEL
LIN {X 0,Y 430.603,Z 1138.835,A -85,B 0,C 180,E1 19874.836,E2 19874.836} C_VEL
LIN {X 0,Y 430.343,Z 1134.363,A -85,B 0,C 180,E1 19873.997,E2 19873.997} C_VEL
LIN {X 0,Y 426.801,Z 1123.94,A -85,B 0,C 180,E1 19872.111,E2 19872.111} C_VEL
LIN {X 0,Y 426.198,Z 1118.718,A -85,B 0,C 180,E1 19871.338,E2 19871.338} C_VEL
LIN {X 0,Y 426.345,Z 1117.094,A -85,B 0,C 180,E1 19871.131,E2 19871.131} C_VEL
LIN {X 0,Y 428.128,Z 1103.64,A -85,B 0,C 180,E1 19869.634,E2 19869.634} C_VEL
LIN {X 0,Y 429.746,Z 1089.223,A -85,B 0,C 180,E1 19868.35,E2 19868.35} C_VEL
LIN {X 0,Y 431.228,Z 1073.046,A -85,B 0,C 180,E1 19867.217,E2 19867.217} C_VEL
LIN {X 0,Y 432.362,Z 1056.491,A -85,B 0,C 180,E1 19866.335,E2 19866.335} C_VEL
LIN {X 0,Y 433.08,Z 1039.349,A -85,B 0,C 180,E1 19865.688,E2 19865.688} C_VEL
LIN {X 0,Y 433.377,Z 1020.394,A -85,B 0,C 180,E1 19865.245,E2 19865.245} C_VEL
LIN {X 0,Y 436.903,Z 864.811,A -85,B 0,C 180,E1 19862.665,E2 19862.665} C_VEL
LIN {X 0,Y 436.333,Z 860.009,A -85,B 0,C 180,E1 19862.535,E2 19862.535} C_VEL
LIN {X 0,Y 439.115,Z 812.632,A -85,B 0,C 180,E1 19858.874,E2 19858.874} C_VEL
LIN {X 0,Y 442.692,Z 763.311,A -85,B 0,C 180,E1 19854.903,E2 19854.903} C_VEL
LIN {X 0,Y 446.313,Z 716.16,A -85,B 0,C 180,E1 19851.065,E2 19851.065} C_VEL
LIN {X 0,Y 446.736,Z 707.626,A -85,B 0,C 180,E1 19850.349,E2 19850.349} C_VEL
LIN {X 0,Y 442.481,Z 693.604,A -85,B 0,C 180,E1 19848.667,E2 19848.667} C_VEL
LIN {X 0,Y 444.297,Z 694.356,A -85,B 0,C 180,E1 19848.401,E2 19848.401} C_VEL
LIN {X 0,Y 447.037,Z 693.608,A -85,B 0,C 180,E1 19848.069,E2 19848.069} C_VEL
LIN {X 0,Y 447.985,Z 693.141,A -85,B 0,C 180,E1 19847.963,E2 19847.963} C_VEL
LIN {X 0,Y 452.007,Z 692.362,A -85,B 0,C 180,E1 19847.482,E2 19847.482} C_VEL
LIN {X 0,Y 452.733,Z 692.943,A -85,B 0,C 180,E1 19847.373,E2 19847.373} C_VEL
LIN {X 0,Y 469.028,Z 716.488,A -85,B 0,C 180,E1 19844.706,E2 19844.706} C_VEL
LIN {X 0,Y 477.176,Z 729.047,A -85,B 0,C 180,E1 19843.441,E2 19843.441} C_VEL
LIN {X 0,Y 458.086,Z 977.833,A -85,B 0,C 180,E1 19838.071,E2 19838.071} C_VEL
LIN {X 0,Y 456.07,Z 1002.053,A -85,B 0,C 180,E1 19837.315,E2 19837.315} C_VEL
LIN {X 0,Y 453.676,Z 1024.069,A -85,B 0,C 180,E1 19836.417,E2 19836.417} C_VEL
LIN {X 0,Y 450.683,Z 1046.307,A -85,B 0,C 180,E1 19835.267,E2 19835.267} C_VEL
LIN {X 0,Y 447.279,Z 1067.874,A -85,B 0,C 180,E1 19833.901,E2 19833.901} C_VEL
LIN {X 0,Y 443.578,Z 1088.971,A -85,B 0,C 180,E1 19832.292,E2 19832.292} C_VEL
LIN {X 0,Y 439.837,Z 1108.473,A -85,B 0,C 180,E1 19830.529,E2 19830.529} C_VEL
LIN {X 0,Y 435.994,Z 1126.862,A -85,B 0,C 180,E1 19828.553,E2 19828.553} C_VEL
LIN {X 0,Y 432.259,Z 1144.216,A -85,B 0,C 180,E1 19826.368,E2 19826.368} C_VEL
LIN {X 0,Y 428.854,Z 1159.813,A -85,B 0,C 180,E1 19824.081,E2 19824.081} C_VEL
LIN {X 0,Y 425.758,Z 1173.967,A -85,B 0,C 180,E1 19821.636,E2 19821.636} C_VEL
LIN {X 0,Y 422.904,Z 1187.457,A -85,B 0,C 180,E1 19818.9,E2 19818.9} C_VEL
LIN {X 0,Y 420.673,Z 1198.946,A -85,B 0,C 180,E1 19816.147,E2 19816.147} C_VEL
LIN {X 0,Y 418.972,Z 1208.525,A -85,B 0,C 180,E1 19813.385,E2 19813.385} C_VEL
LIN {X 0,Y 417.675,Z 1217.199,A -85,B 0,C 180,E1 19810.343,E2 19810.343} C_VEL
LIN {X 0,Y 416.905,Z 1223.855,A -85,B 0,C 180,E1 19807.441,E2 19807.441} C_VEL
LIN {X 0,Y 416.447,Z 1229.032,A -85,B 0,C 180,E1 19804.407,E2 19804.407} C_VEL
LIN {X 0,Y 416.259,Z 1232.815,A -85,B 0,C 180,E1 19801.239,E2 19801.239} C_VEL
LIN {X 0,Y 416.222,Z 1234.728,A -85,B 0,C 180,E1 19798.486,E2 19798.486} C_VEL
LIN {X 0,Y 416.25,Z 1235.378,A -85,B 0,C 180,E1 19795.453,E2 19795.453} C_VEL
LIN {X 0,Y 416.401,Z 1234.641,A -85,B 0,C 180,E1 19792.55,E2 19792.55} C_VEL
LIN {X 0,Y 416.714,Z 1232.297,A -85,B 0,C 180,E1 19789.493,E2 19789.493} C_VEL
LIN {X 0,Y 417.395,Z 1228.258,A -85,B 0,C 180,E1 19786.281,E2 19786.281} C_VEL
LIN {X 0,Y 418.527,Z 1222.792,A -85,B 0,C 180,E1 19783.197,E2 19783.197} C_VEL
LIN {X 0,Y 420.267,Z 1215.487,A -85,B 0,C 180,E1 19780.109,E2 19780.109} C_VEL
LIN {X 0,Y 422.584,Z 1206.804,A -85,B 0,C 180,E1 19777.167,E2 19777.167} C_VEL
LIN {X 0,Y 425.466,Z 1196.828,A -85,B 0,C 180,E1 19774.379,E2 19774.379} C_VEL
LIN {X 0,Y 429.055,Z 1184.876,A -85,B 0,C 180,E1 19771.614,E2 19771.614} C_VEL
LIN {X 0,Y 432.885,Z 1172.111,A -85,B 0,C 180,E1 19769.151,E2 19769.151} C_VEL
LIN {X 0,Y 437.062,Z 1158.089,A -85,B 0,C 180,E1 19766.854,E2 19766.854} C_VEL
LIN {X 0,Y 441.479,Z 1142.748,A -85,B 0,C 180,E1 19764.722,E2 19764.722} C_VEL
LIN {X 0,Y 446.067,Z 1125.754,A -85,B 0,C 180,E1 19762.729,E2 19762.729} C_VEL
LIN {X 0,Y 450.601,Z 1107.493,A -85,B 0,C 180,E1 19760.935,E2 19760.935} C_VEL
LIN {X 0,Y 454.96,Z 1087.835,A -85,B 0,C 180,E1 19759.335,E2 19759.335} C_VEL
LIN {X 0,Y 458.776,Z 1068.017,A -85,B 0,C 180,E1 19758.002,E2 19758.002} C_VEL
LIN {X 0,Y 462.175,Z 1047.307,A -85,B 0,C 180,E1 19756.87,E2 19756.87} C_VEL
LIN {X 0,Y 465.147,Z 1025.476,A -85,B 0,C 180,E1 19755.919,E2 19755.919} C_VEL
LIN {X 0,Y 469.07,Z 999.645,A -85,B 0,C 180,E1 19754.994,E2 19754.994} C_VEL
LIN {X 0,Y 475.185,Z 973.419,A -85,B 0,C 180,E1 19754.127,E2 19754.127} C_VEL
LIN {X 0,Y 479.438,Z 958.857,A -85,B 0,C 180,E1 19753.667,E2 19753.667} C_VEL
LIN {X 0,Y 473.669,Z 977.944,A -85,B 0,C 180,E1 19753.154,E2 19753.154} C_VEL
LIN {X 0,Y 468.025,Z 996.864,A -85,B 0,C 180,E1 19752.381,E2 19752.381} C_VEL
LIN {X 0,Y 457.711,Z 1033.651,A -85,B 0,C 180,E1 19750.516,E2 19750.516} C_VEL
LIN {X 0,Y 449.631,Z 1065.505,A -85,B 0,C 180,E1 19748.594,E2 19748.594} C_VEL
LIN {X 0,Y 442.378,Z 1097.751,A -85,B 0,C 180,E1 19746.314,E2 19746.314} C_VEL
LIN {X 0,Y 436.36,Z 1127.864,A -85,B 0,C 180,E1 19743.838,E2 19743.838} C_VEL
LIN {X 0,Y 431.261,Z 1156.373,A -85,B 0,C 180,E1 19741.135,E2 19741.135} C_VEL
LIN {X 0,Y 427.366,Z 1180.45,A -85,B 0,C 180,E1 19738.51,E2 19738.51} C_VEL
LIN {X 0,Y 424.286,Z 1200.903,A -85,B 0,C 180,E1 19735.924,E2 19735.924} C_VEL
LIN {X 0,Y 421.814,Z 1218.634,A -85,B 0,C 180,E1 19733.322,E2 19733.322} C_VEL
LIN {X 0,Y 419.92,Z 1233.425,A -85,B 0,C 180,E1 19730.782,E2 19730.782} C_VEL
LIN {X 0,Y 418.471,Z 1246.005,A -85,B 0,C 180,E1 19728.242,E2 19728.242} C_VEL
LIN {X 0,Y 417.405,Z 1257.063,A -85,B 0,C 180,E1 19725.565,E2 19725.565} C_VEL
LIN {X 0,Y 416.696,Z 1266.009,A -85,B 0,C 180,E1 19722.896,E2 19722.896} C_VEL
LIN {X 0,Y 416.32,Z 1273.074,A -85,B 0,C 180,E1 19720.239,E2 19720.239} C_VEL
LIN {X 0,Y 416.166,Z 1278.632,A -85,B 0,C 180,E1 19717.456,E2 19717.456} C_VEL
LIN {X 0,Y 416.157,Z 1282.226,A -85,B 0,C 180,E1 19714.826,E2 19714.826} C_VEL
LIN {X 0,Y 416.189,Z 1284.249,A -85,B 0,C 180,E1 19712.205,E2 19712.205} C_VEL
LIN {X 0,Y 416.208,Z 1284.72,A -85,B 0,C 180,E1 19709.589,E2 19709.589} C_VEL
LIN {X 0,Y 416.188,Z 1283.581,A -85,B 0,C 180,E1 19706.834,E2 19706.834} C_VEL
LIN {X 0,Y 416.16,Z 1280.65,A -85,B 0,C 180,E1 19703.934,E2 19703.934} C_VEL
LIN {X 0,Y 416.204,Z 1276.214,A -85,B 0,C 180,E1 19701.157,E2 19701.157} C_VEL
LIN {X 0,Y 416.475,Z 1269.717,A -85,B 0,C 180,E1 19698.227,E2 19698.227} C_VEL
LIN {X 0,Y 417.08,Z 1261.373,A -85,B 0,C 180,E1 19695.281,E2 19695.281} C_VEL
LIN {X 0,Y 418.141,Z 1250.994,A -85,B 0,C 180,E1 19692.323,E2 19692.323} C_VEL
LIN {X 0,Y 419.775,Z 1238.528,A -85,B 0,C 180,E1 19689.36,E2 19689.36} C_VEL
LIN {X 0,Y 422.073,Z 1223.7,A -85,B 0,C 180,E1 19686.402,E2 19686.402} C_VEL
LIN {X 0,Y 424.787,Z 1208.055,A -85,B 0,C 180,E1 19683.737,E2 19683.737} C_VEL
LIN {X 0,Y 428.193,Z 1190.063,A -85,B 0,C 180,E1 19681.097,E2 19681.097} C_VEL
LIN {X 0,Y 432.337,Z 1169.327,A -85,B 0,C 180,E1 19678.49,E2 19678.49} C_VEL
LIN {X 0,Y 437.013,Z 1146.689,A -85,B 0,C 180,E1 19676.066,E2 19676.066} C_VEL
LIN {X 0,Y 441.698,Z 1124.257,A -85,B 0,C 180,E1 19674.027,E2 19674.027} C_VEL
LIN {X 0,Y 446.861,Z 1099.599,A -85,B 0,C 180,E1 19672.108,E2 19672.108} C_VEL
LIN {X 0,Y 451.591,Z 1076.642,A -85,B 0,C 180,E1 19670.601,E2 19670.601} C_VEL
LIN {X 0,Y 456.711,Z 1050.875,A -85,B 0,C 180,E1 19669.196,E2 19669.196} C_VEL
LIN {X 0,Y 461.121,Z 1027.399,A -85,B 0,C 180,E1 19668.142,E2 19668.142} C_VEL
LIN {X 0,Y 465.401,Z 1001.448,A -85,B 0,C 180,E1 19667.213,E2 19667.213} C_VEL
LIN {X 0,Y 468.904,Z 975.996,A -85,B 0,C 180,E1 19666.486,E2 19666.486} C_VEL
LIN {X 0,Y 471.857,Z 956.638,A -85,B 0,C 180,E1 19666.134,E2 19666.134} C_VEL
LIN {X 0,Y 462.994,Z 937.246,A -85,B 0,C 180,E1 19664.687,E2 19664.687} C_VEL
LIN {X 0,Y 457.374,Z 921.837,A -85,B 0,C 180,E1 19663.609,E2 19663.609} C_VEL
LIN {X 0,Y 455.663,Z 901.467,A -85,B 0,C 180,E1 19661.171,E2 19661.171} C_VEL
LIN {X 0,Y 456.464,Z 878.083,A -85,B 0,C 180,E1 19658.559,E2 19658.559} C_VEL
LIN {X 0,Y 465.212,Z 822.605,A -85,B 0,C 180,E1 19652.824,E2 19652.824} C_VEL
LIN {X 0,Y 471.162,Z 789.246,A -85,B 0,C 180,E1 19649.355,E2 19649.355} C_VEL
LIN {X 0,Y 475.744,Z 763.955,A -85,B 0,C 180,E1 19646.669,E2 19646.669} C_VEL
LIN {X 0,Y 468.812,Z 745.975,A -85,B 0,C 180,E1 19643.372,E2 19643.372} C_VEL
LIN {X 0,Y 461.931,Z 728.921,A -85,B 0,C 180,E1 19639.999,E2 19639.999} C_VEL
LIN {X 0,Y 455.199,Z 713.051,A -85,B 0,C 180,E1 19636.592,E2 19636.592} C_VEL
LIN {X 0,Y 448.84,Z 698.792,A -85,B 0,C 180,E1 19633.265,E2 19633.265} C_VEL
LIN {X 0,Y 442.735,Z 685.312,A -85,B 0,C 180,E1 19629.883,E2 19629.883} C_VEL
LIN {X 0,Y 436.312,Z 671.841,A -85,B 0,C 180,E1 19626.183,E2 19626.183} C_VEL
LIN {X 0,Y 431.523,Z 662.222,A -85,B 0,C 180,E1 19623.321,E2 19623.321} C_VEL
LIN {X 0,Y 429.372,Z 657.95,A -85,B 0,C 180,E1 19622.002,E2 19622.002} C_VEL
LIN {X 0,Y 427.367,Z 653.801,A -85,B 0,C 180,E1 19620.67,E2 19620.67} C_VEL
LIN {X 0,Y 424.981,Z 649.12,A -85,B 0,C 180,E1 19619.137,E2 19619.137} C_VEL
LIN {X 0,Y 422.918,Z 644.904,A -85,B 0,C 180,E1 19617.696,E2 19617.696} C_VEL
LIN {X 0,Y 421.113,Z 641.336,A -85,B 0,C 180,E1 19616.461,E2 19616.461} C_VEL
LIN {X 0,Y 418.691,Z 636.714,A -85,B 0,C 180,E1 19614.749,E2 19614.749} C_VEL
LIN {X 0,Y 418.539,Z 635.844,A -85,B 0,C 180,E1 19614.448,E2 19614.448} C_VEL
LIN {X 0,Y 418.533,Z 635.841,A -85,B 0,C 180,E1 19610.651,E2 19610.651} C_VEL
LIN {X 0,Y 418.544,Z 635.832,A -85,B 0,C 180,E1 19606.742,E2 19606.742} C_VEL
LIN {X 0,Y 418.539,Z 635.834,A -85,B 0,C 180,E1 19602.911,E2 19602.911} C_VEL
LIN {X 0,Y 418.535,Z 635.839,A -85,B 0,C 180,E1 19599.077,E2 19599.077} C_VEL
LIN {X 0,Y 418.548,Z 635.843,A -85,B 0,C 180,E1 19595.136,E2 19595.136} C_VEL
LIN {X 0,Y 418.539,Z 635.847,A -85,B 0,C 180,E1 19591.146,E2 19591.146} C_VEL
LIN {X 0,Y 418.543,Z 635.846,A -85,B 0,C 180,E1 19587.233,E2 19587.233} C_VEL
LIN {X 0,Y 418.537,Z 635.848,A -85,B 0,C 180,E1 19583.326,E2 19583.326} C_VEL
LIN {X 0,Y 418.549,Z 635.847,A -85,B 0,C 180,E1 19579.433,E2 19579.433} C_VEL
LIN {X 0,Y 418.561,Z 636.009,A -85,B 0,C 180,E1 19576.461,E2 19576.461} C_VEL
LIN {X 0,Y 420.007,Z 639.514,A -85,B 0,C 180,E1 19575.96,E2 19575.96} C_VEL
LIN {X 0,Y 427.692,Z 656.136,A -85,B 0,C 180,E1 19573.552,E2 19573.552} C_VEL
LIN {X 0,Y 435.336,Z 675.008,A -85,B 0,C 180,E1 19571.027,E2 19571.027} C_VEL
LIN {X 0,Y 442.291,Z 695.322,A -85,B 0,C 180,E1 19568.537,E2 19568.537} C_VEL
LIN {X 0,Y 445.445,Z 706.919,A -85,B 0,C 180,E1 19567.214,E2 19567.214} C_VEL
LIN {X 0,Y 442.185,Z 750.908,A -85,B 0,C 180,E1 19563.64,E2 19563.64} C_VEL
LIN {X 0,Y 438.785,Z 798.693,A -85,B 0,C 180,E1 19559.784,E2 19559.784} C_VEL
LIN {X 0,Y 435.887,Z 846.528,A -85,B 0,C 180,E1 19556.056,E2 19556.056} C_VEL
LIN {X 0,Y 435.299,Z 860.608,A -85,B 0,C 180,E1 19555.027,E2 19555.027} C_VEL
LIN {X 0,Y 435.818,Z 867.793,A -85,B 0,C 180,E1 19554.864,E2 19554.864} C_VEL
LIN {X 0,Y 432.245,Z 1026.924,A -85,B 0,C 180,E1 19552.221,E2 19552.221} C_VEL
LIN {X 0,Y 431.829,Z 1044.795,A -85,B 0,C 180,E1 19551.72,E2 19551.72} C_VEL
LIN {X 0,Y 431.024,Z 1061.75,A -85,B 0,C 180,E1 19551,E2 19551} C_VEL
LIN {X 0,Y 429.868,Z 1077.837,A -85,B 0,C 180,E1 19550.063,E2 19550.063} C_VEL
LIN {X 0,Y 428.449,Z 1092.895,A -85,B 0,C 180,E1 19548.926,E2 19548.926} C_VEL
LIN {X 0,Y 426.81,Z 1107.467,A -85,B 0,C 180,E1 19547.544,E2 19547.544} C_VEL
LIN {X 0,Y 425.094,Z 1120.817,A -85,B 0,C 180,E1 19545.972,E2 19545.972} C_VEL
LIN {X 0,Y 423.389,Z 1132.802,A -85,B 0,C 180,E1 19544.216,E2 19544.216} C_VEL
LIN {X 0,Y 421.816,Z 1143.292,A -85,B 0,C 180,E1 19542.316,E2 19542.316} C_VEL
LIN {X 0,Y 420.445,Z 1152.343,A -85,B 0,C 180,E1 19540.272,E2 19540.272} C_VEL
LIN {X 0,Y 419.325,Z 1159.918,A -85,B 0,C 180,E1 19538.086,E2 19538.086} C_VEL
LIN {X 0,Y 418.482,Z 1165.882,A -85,B 0,C 180,E1 19535.757,E2 19535.757} C_VEL
LIN {X 0,Y 417.92,Z 1170.217,A -85,B 0,C 180,E1 19533.29,E2 19533.29} C_VEL
LIN {X 0,Y 417.659,Z 1172.571,A -85,B 0,C 180,E1 19530.958,E2 19530.958} C_VEL
LIN {X 0,Y 417.599,Z 1173.237,A -85,B 0,C 180,E1 19528.489,E2 19528.489} C_VEL
LIN {X 0,Y 417.768,Z 1172.117,A -85,B 0,C 180,E1 19526.018,E2 19526.018} C_VEL
LIN {X 0,Y 418.202,Z 1169.186,A -85,B 0,C 180,E1 19523.546,E2 19523.546} C_VEL
LIN {X 0,Y 418.908,Z 1164.49,A -85,B 0,C 180,E1 19521.183,E2 19521.183} C_VEL
LIN {X 0,Y 419.98,Z 1157.719,A -85,B 0,C 180,E1 19518.783,E2 19518.783} C_VEL
LIN {X 0,Y 421.265,Z 1149.92,A -85,B 0,C 180,E1 19516.687,E2 19516.687} C_VEL
LIN {X 0,Y 422.848,Z 1140.197,A -85,B 0,C 180,E1 19514.641,E2 19514.641} C_VEL
LIN {X 0,Y 424.624,Z 1128.875,A -85,B 0,C 180,E1 19512.739,E2 19512.739} C_VEL
LIN {X 0,Y 426.345,Z 1117.094,A -85,B 0,C 180,E1 19511.131,E2 19511.131} C_VEL
LIN {X 0,Y 426.22,Z 1111.509,A -85,B 0,C 180,E1 19510.404,E2 19510.404} C_VEL
LIN {X 0,Y 423.037,Z 1099.556,A -85,B 0,C 180,E1 19508.872,E2 19508.872} C_VEL
LIN {X 0,Y 422.19,Z 1092.478,A -85,B 0,C 180,E1 19508.153,E2 19508.153} C_VEL
LIN {X 0,Y 422.298,Z 1090.589,A -85,B 0,C 180,E1 19507.996,E2 19507.996} C_VEL
LIN {X 0,Y 423.806,Z 1074.881,A -85,B 0,C 180,E1 19506.868,E2 19506.868} C_VEL
LIN {X 0,Y 425.017,Z 1058.022,A -85,B 0,C 180,E1 19505.945,E2 19505.945} C_VEL
LIN {X 0,Y 425.79,Z 1041.036,A -85,B 0,C 180,E1 19505.281,E2 19505.281} C_VEL
LIN {X 0,Y 426.107,Z 1022.498,A -85,B 0,C 180,E1 19504.829,E2 19504.829} C_VEL
LIN {X 0,Y 429.795,Z 865.75,A -85,B 0,C 180,E1 19502.188,E2 19502.188} C_VEL
LIN {X 0,Y 429.244,Z 860.762,A -85,B 0,C 180,E1 19502.042,E2 19502.042} C_VEL
LIN {X 0,Y 432.139,Z 813.728,A -85,B 0,C 180,E1 19498.374,E2 19498.374} C_VEL
LIN {X 0,Y 435.786,Z 765.129,A -85,B 0,C 180,E1 19494.432,E2 19494.432} C_VEL
LIN {X 0,Y 439.589,Z 717.465,A -85,B 0,C 180,E1 19490.523,E2 19490.523} C_VEL
LIN {X 0,Y 439.943,Z 710.808,A -85,B 0,C 180,E1 19489.968,E2 19489.968} C_VEL
LIN {X 0,Y 437.612,Z 702.712,A -85,B 0,C 180,E1 19488.978,E2 19488.978} C_VEL
LIN {X 0,Y 439.45,Z 703.454,A -85,B 0,C 180,E1 19488.711,E2 19488.711} C_VEL
LIN {X 0,Y 442.233,Z 702.683,A -85,B 0,C 180,E1 19488.38,E2 19488.38} C_VEL
LIN {X 0,Y 443.187,Z 702.217,A -85,B 0,C 180,E1 19488.273,E2 19488.273} C_VEL
LIN {X 0,Y 447.183,Z 701.391,A -85,B 0,C 180,E1 19487.784,E2 19487.784} C_VEL
LIN {X 0,Y 449.578,Z 700.842,A -85,B 0,C 180,E1 19487.501,E2 19487.501} C_VEL
LIN {X 0,Y 466.167,Z 724.983,A -85,B 0,C 180,E1 19484.766,E2 19484.766} C_VEL
LIN {X 0,Y 470.899,Z 732.548,A -85,B 0,C 180,E1 19484.012,E2 19484.012} C_VEL
LIN {X 0,Y 451.252,Z 978.328,A -85,B 0,C 180,E1 19478.591,E2 19478.591} C_VEL
LIN {X 0,Y 449.171,Z 1002.675,A -85,B 0,C 180,E1 19477.823,E2 19477.823} C_VEL
LIN {X 0,Y 446.697,Z 1024.798,A -85,B 0,C 180,E1 19476.907,E2 19476.907} C_VEL
LIN {X 0,Y 443.731,Z 1046.221,A -85,B 0,C 180,E1 19475.784,E2 19475.784} C_VEL
LIN {X 0,Y 440.317,Z 1067.451,A -85,B 0,C 180,E1 19474.433,E2 19474.433} C_VEL
LIN {X 0,Y 436.656,Z 1087.971,A -85,B 0,C 180,E1 19472.868,E2 19472.868} C_VEL
LIN {X 0,Y 432.793,Z 1107.522,A -85,B 0,C 180,E1 19471.088,E2 19471.088} C_VEL
LIN {X 0,Y 428.835,Z 1126.124,A -85,B 0,C 180,E1 19469.088,E2 19469.088} C_VEL
LIN {X 0,Y 424.83,Z 1144.273,A -85,B 0,C 180,E1 19466.79,E2 19466.79} C_VEL
LIN {X 0,Y 421.218,Z 1160.378,A -85,B 0,C 180,E1 19464.396,E2 19464.396} C_VEL
LIN {X 0,Y 417.941,Z 1174.958,A -85,B 0,C 180,E1 19461.832,E2 19461.832} C_VEL
LIN {X 0,Y 415.092,Z 1188.047,A -85,B 0,C 180,E1 19459.123,E2 19459.123} C_VEL
LIN {X 0,Y 412.794,Z 1199.546,A -85,B 0,C 180,E1 19456.319,E2 19456.319} C_VEL
LIN {X 0,Y 411.042,Z 1209.128,A -85,B 0,C 180,E1 19453.505,E2 19453.505} C_VEL
LIN {X 0,Y 409.709,Z 1217.8,A -85,B 0,C 180,E1 19450.405,E2 19450.405} C_VEL
LIN {X 0,Y 408.919,Z 1224.451,A -85,B 0,C 180,E1 19447.446,E2 19447.446} C_VEL
LIN {X 0,Y 408.468,Z 1229.413,A -85,B 0,C 180,E1 19444.493,E2 19444.493} C_VEL
LIN {X 0,Y 408.279,Z 1233.149,A -85,B 0,C 180,E1 19441.403,E2 19441.403} C_VEL
LIN {X 0,Y 408.236,Z 1235.216,A -85,B 0,C 180,E1 19438.456,E2 19438.456} C_VEL
LIN {X 0,Y 408.272,Z 1235.932,A -85,B 0,C 180,E1 19435.364,E2 19435.364} C_VEL
LIN {X 0,Y 408.438,Z 1235.234,A -85,B 0,C 180,E1 19432.403,E2 19432.403} C_VEL
LIN {X 0,Y 408.788,Z 1232.956,A -85,B 0,C 180,E1 19429.287,E2 19429.287} C_VEL
LIN {X 0,Y 409.533,Z 1228.989,A -85,B 0,C 180,E1 19426.012,E2 19426.012} C_VEL
LIN {X 0,Y 410.765,Z 1223.586,A -85,B 0,C 180,E1 19422.87,E2 19422.87} C_VEL
LIN {X 0,Y 412.687,Z 1216.213,A -85,B 0,C 180,E1 19419.664,E2 19419.664} C_VEL
LIN {X 0,Y 415.263,Z 1207.329,A -85,B 0,C 180,E1 19416.591,E2 19416.591} C_VEL
LIN {X 0,Y 418.544,Z 1196.794,A -85,B 0,C 180,E1 19413.618,E2 19413.618} C_VEL
LIN {X 0,Y 422.328,Z 1185.14,A -85,B 0,C 180,E1 19410.886,E2 19410.886} C_VEL
LIN {X 0,Y 426.822,Z 1171.279,A -85,B 0,C 180,E1 19408.191,E2 19408.191} C_VEL
LIN {X 0,Y 431.38,Z 1156.838,A -85,B 0,C 180,E1 19405.843,E2 19405.843} C_VEL
LIN {X 0,Y 436.037,Z 1141.472,A -85,B 0,C 180,E1 19403.727,E2 19403.727} C_VEL
LIN {X 0,Y 440.915,Z 1124.457,A -85,B 0,C 180,E1 19401.749,E2 19401.749} C_VEL
LIN {X 0,Y 445.645,Z 1106.523,A -85,B 0,C 180,E1 19399.997,E2 19399.997} C_VEL
LIN {X 0,Y 450.076,Z 1087.931,A -85,B 0,C 180,E1 19398.478,E2 19398.478} C_VEL
LIN {X 0,Y 454.223,Z 1068.259,A -85,B 0,C 180,E1 19397.14,E2 19397.14} C_VEL
LIN {X 0,Y 458.152,Z 1047.054,A -85,B 0,C 180,E1 19395.964,E2 19395.964} C_VEL
LIN {X 0,Y 461.989,Z 1023.681,A -85,B 0,C 180,E1 19394.927,E2 19394.927} C_VEL
LIN {X 0,Y 466.702,Z 1001.184,A -85,B 0,C 180,E1 19394.078,E2 19394.078} C_VEL
LIN {X 0,Y 469.633,Z 990.52,A -85,B 0,C 180,E1 19393.692,E2 19393.692} C_VEL
LIN {X 0,Y 458.725,Z 1023.589,A -85,B 0,C 180,E1 19392.089,E2 19392.089} C_VEL
LIN {X 0,Y 449.213,Z 1054.514,A -85,B 0,C 180,E1 19390.288,E2 19390.288} C_VEL
LIN {X 0,Y 440.552,Z 1085.799,A -85,B 0,C 180,E1 19388.124,E2 19388.124} C_VEL
LIN {X 0,Y 432.993,Z 1116.622,A -85,B 0,C 180,E1 19385.624,E2 19385.624} C_VEL
LIN {X 0,Y 426.689,Z 1146.266,A -85,B 0,C 180,E1 19382.855,E2 19382.855} C_VEL
LIN {X 0,Y 421.73,Z 1172.612,A -85,B 0,C 180,E1 19380.019,E2 19380.019} C_VEL
LIN {X 0,Y 417.951,Z 1194.785,A -85,B 0,C 180,E1 19377.273,E2 19377.273} C_VEL
LIN {X 0,Y 415.083,Z 1213.147,A -85,B 0,C 180,E1 19374.63,E2 19374.63} C_VEL
LIN {X 0,Y 412.848,Z 1228.554,A -85,B 0,C 180,E1 19372.051,E2 19372.051} C_VEL
LIN {X 0,Y 411.154,Z 1241.735,A -85,B 0,C 180,E1 19369.463,E2 19369.463} C_VEL
LIN {X 0,Y 409.827,Z 1253.414,A -85,B 0,C 180,E1 19366.734,E2 19366.734} C_VEL
LIN {X 0,Y 408.948,Z 1263.002,A -85,B 0,C 180,E1 19364.01,E2 19364.01} C_VEL
LIN {X 0,Y 408.435,Z 1270.66,A -85,B 0,C 180,E1 19361.296,E2 19361.296} C_VEL
LIN {X 0,Y 408.206,Z 1276.518,A -85,B 0,C 180,E1 19358.595,E2 19358.595} C_VEL
LIN {X 0,Y 408.157,Z 1280.655,A -85,B 0,C 180,E1 19355.907,E2 19355.907} C_VEL
LIN {X 0,Y 408.191,Z 1283.188,A -85,B 0,C 180,E1 19353.232,E2 19353.232} C_VEL
LIN {X 0,Y 408.227,Z 1284.177,A -85,B 0,C 180,E1 19350.423,E2 19350.423} C_VEL
LIN {X 0,Y 408.213,Z 1283.502,A -85,B 0,C 180,E1 19347.615,E2 19347.615} C_VEL
LIN {X 0,Y 408.182,Z 1281.19,A -85,B 0,C 180,E1 19344.802,E2 19344.802} C_VEL
LIN {X 0,Y 408.188,Z 1277.186,A -85,B 0,C 180,E1 19341.976,E2 19341.976} C_VEL
LIN {X 0,Y 408.388,Z 1271.211,A -85,B 0,C 180,E1 19338.992,E2 19338.992} C_VEL
LIN {X 0,Y 408.864,Z 1263.797,A -85,B 0,C 180,E1 19336.136,E2 19336.136} C_VEL
LIN {X 0,Y 409.836,Z 1253.654,A -85,B 0,C 180,E1 19333.015,E2 19333.015} C_VEL
LIN {X 0,Y 411.292,Z 1242.221,A -85,B 0,C 180,E1 19330.104,E2 19330.104} C_VEL
LIN {X 0,Y 413.427,Z 1228.131,A -85,B 0,C 180,E1 19327.086,E2 19327.086} C_VEL
LIN {X 0,Y 416.16,Z 1212.369,A -85,B 0,C 180,E1 19324.225,E2 19324.225} C_VEL
LIN {X 0,Y 419.446,Z 1195.071,A -85,B 0,C 180,E1 19321.528,E2 19321.528} C_VEL
LIN {X 0,Y 423.491,Z 1175.175,A -85,B 0,C 180,E1 19318.867,E2 19318.867} C_VEL
LIN {X 0,Y 428.218,Z 1152.866,A -85,B 0,C 180,E1 19316.322,E2 19316.322} C_VEL
LIN {X 0,Y 433.445,Z 1128.469,A -85,B 0,C 180,E1 19313.97,E2 19313.97} C_VEL
LIN {X 0,Y 438.037,Z 1107.331,A -85,B 0,C 180,E1 19312.229,E2 19312.229} C_VEL
LIN {X 0,Y 443.457,Z 1081.817,A -85,B 0,C 180,E1 19310.437,E2 19310.437} C_VEL
LIN {X 0,Y 448.417,Z 1058.007,A -85,B 0,C 180,E1 19309.04,E2 19309.04} C_VEL
LIN {X 0,Y 453.329,Z 1032.978,A -85,B 0,C 180,E1 19307.84,E2 19307.84} C_VEL
LIN {X 0,Y 457.967,Z 1007.184,A -85,B 0,C 180,E1 19306.834,E2 19306.834} C_VEL
LIN {X 0,Y 461.698,Z 981.087,A -85,B 0,C 180,E1 19306.031,E2 19306.031} C_VEL
LIN {X 0,Y 465.062,Z 959.112,A -85,B 0,C 180,E1 19305.571,E2 19305.571} C_VEL
LIN {X 0,Y 456.564,Z 939.704,A -85,B 0,C 180,E1 19304.12,E2 19304.12} C_VEL
LIN {X 0,Y 449.819,Z 920.721,A -85,B 0,C 180,E1 19302.794,E2 19302.794} C_VEL
LIN {X 0,Y 449.425,Z 918.369,A -85,B 0,C 180,E1 19302.559,E2 19302.559} C_VEL
LIN {X 0,Y 448.517,Z 896.977,A -85,B 0,C 180,E1 19300.028,E2 19300.028} C_VEL
LIN {X 0,Y 450.346,Z 872.509,A -85,B 0,C 180,E1 19297.311,E2 19297.311} C_VEL
LIN {X 0,Y 458.039,Z 827.434,A -85,B 0,C 180,E1 19292.629,E2 19292.629} C_VEL
LIN {X 0,Y 464.151,Z 794.048,A -85,B 0,C 180,E1 19289.134,E2 19289.134} C_VEL
LIN {X 0,Y 469.065,Z 767.681,A -85,B 0,C 180,E1 19286.32,E2 19286.32} C_VEL
LIN {X 0,Y 462.306,Z 750.051,A -85,B 0,C 180,E1 19283.046,E2 19283.046} C_VEL
LIN {X 0,Y 455.646,Z 733.419,A -85,B 0,C 180,E1 19279.716,E2 19279.716} C_VEL
LIN {X 0,Y 449.02,Z 717.663,A -85,B 0,C 180,E1 19276.295,E2 19276.295} C_VEL
LIN {X 0,Y 442.042,Z 701.823,A -85,B 0,C 180,E1 19272.542,E2 19272.542} C_VEL
LIN {X 0,Y 435.86,Z 688.497,A -85,B 0,C 180,E1 19269.108,E2 19269.108} C_VEL
LIN {X 0,Y 430.58,Z 677.263,A -85,B 0,C 180,E1 19265.998,E2 19265.998} C_VEL
LIN {X 0,Y 425.58,Z 667.158,A -85,B 0,C 180,E1 19262.963,E2 19262.963} C_VEL
LIN {X 0,Y 421.956,Z 659.669,A -85,B 0,C 180,E1 19260.594,E2 19260.594} C_VEL
LIN {X 0,Y 419.136,Z 654.264,A -85,B 0,C 180,E1 19258.77,E2 19258.77} C_VEL
LIN {X 0,Y 417.332,Z 650.525,A -85,B 0,C 180,E1 19257.497,E2 19257.497} C_VEL
LIN {X 0,Y 415.006,Z 645.902,A -85,B 0,C 180,E1 19255.855,E2 19255.855} C_VEL
LIN {X 0,Y 413.228,Z 642.482,A -85,B 0,C 180,E1 19254.585,E2 19254.585} C_VEL
LIN {X 0,Y 412.417,Z 640.991,A -85,B 0,C 180,E1 19254.016,E2 19254.016} C_VEL
LIN {X 0,Y 410.752,Z 637.618,A -85,B 0,C 180,E1 19252.728,E2 19252.728} C_VEL
LIN {X 0,Y 410.609,Z 636.821,A -85,B 0,C 180,E1 19252.444,E2 19252.444} C_VEL
LIN {X 0,Y 410.594,Z 636.833,A -85,B 0,C 180,E1 19248.481,E2 19248.481} C_VEL
LIN {X 0,Y 410.606,Z 636.833,A -85,B 0,C 180,E1 19244.607,E2 19244.607} C_VEL
LIN {X 0,Y 410.606,Z 636.825,A -85,B 0,C 180,E1 19240.659,E2 19240.659} C_VEL
LIN {X 0,Y 410.598,Z 636.822,A -85,B 0,C 180,E1 19236.765,E2 19236.765} C_VEL
LIN {X 0,Y 410.594,Z 636.819,A -85,B 0,C 180,E1 19232.91,E2 19232.91} C_VEL
LIN {X 0,Y 410.603,Z 636.818,A -85,B 0,C 180,E1 19228.918,E2 19228.918} C_VEL
LIN {X 0,Y 410.598,Z 636.817,A -85,B 0,C 180,E1 19225.091,E2 19225.091} C_VEL
LIN {X 0,Y 410.601,Z 636.82,A -85,B 0,C 180,E1 19221.189,E2 19221.189} C_VEL
LIN {X 0,Y 410.615,Z 636.943,A -85,B 0,C 180,E1 19217.393,E2 19217.393} C_VEL
LIN {X 0,Y 411.704,Z 639.961,A -85,B 0,C 180,E1 19216.964,E2 19216.964} C_VEL
LIN {X 0,Y 413.004,Z 642.456,A -85,B 0,C 180,E1 19216.562,E2 19216.562} C_VEL
LIN {X 0,Y 420.212,Z 657.83,A -85,B 0,C 180,E1 19214.256,E2 19214.256} C_VEL
LIN {X 0,Y 426.995,Z 674.234,A -85,B 0,C 180,E1 19211.97,E2 19211.97} C_VEL
LIN {X 0,Y 433.805,Z 693.285,A -85,B 0,C 180,E1 19209.556,E2 19209.556} C_VEL
LIN {X 0,Y 438.571,Z 709.206,A -85,B 0,C 180,E1 19207.66,E2 19207.66} C_VEL
LIN {X 0,Y 435.281,Z 751.703,A -85,B 0,C 180,E1 19204.175,E2 19204.175} C_VEL
LIN {X 0,Y 431.802,Z 799.284,A -85,B 0,C 180,E1 19200.316,E2 19200.316} C_VEL
LIN {X 0,Y 428.788,Z 846.492,A -85,B 0,C 180,E1 19196.595,E2 19196.595} C_VEL
LIN {X 0,Y 428.102,Z 861.325,A -85,B 0,C 180,E1 19195.493,E2 19195.493} C_VEL
LIN {X 0,Y 428.628,Z 868.686,A -85,B 0,C 180,E1 19195.321,E2 19195.321} C_VEL
LIN {X 0,Y 424.92,Z 1027.546,A -85,B 0,C 180,E1 19192.643,E2 19192.643} C_VEL
LIN {X 0,Y 424.496,Z 1045.301,A -85,B 0,C 180,E1 19192.143,E2 19192.143} C_VEL
LIN {X 0,Y 423.67,Z 1062.205,A -85,B 0,C 180,E1 19191.419,E2 19191.419} C_VEL
LIN {X 0,Y 422.518,Z 1077.959,A -85,B 0,C 180,E1 19190.5,E2 19190.5} C_VEL
LIN {X 0,Y 421.041,Z 1093.184,A -85,B 0,C 180,E1 19189.345,E2 19189.345} C_VEL
LIN {X 0,Y 419.303,Z 1108.114,A -85,B 0,C 180,E1 19187.914,E2 19187.914} C_VEL
LIN {X 0,Y 417.546,Z 1121.32,A -85,B 0,C 180,E1 19186.34,E2 19186.34} C_VEL
LIN {X 0,Y 415.83,Z 1133.004,A -85,B 0,C 180,E1 19184.622,E2 19184.622} C_VEL
LIN {X 0,Y 414.172,Z 1143.624,A -85,B 0,C 180,E1 19182.689,E2 19182.689} C_VEL
LIN {X 0,Y 412.718,Z 1152.789,A -85,B 0,C 180,E1 19180.608,E2 19180.608} C_VEL
LIN {X 0,Y 411.526,Z 1160.491,A -85,B 0,C 180,E1 19178.381,E2 19178.381} C_VEL
LIN {X 0,Y 410.625,Z 1166.569,A -85,B 0,C 180,E1 19176.008,E2 19176.008} C_VEL
LIN {X 0,Y 410.014,Z 1170.988,A -85,B 0,C 180,E1 19173.493,E2 19173.493} C_VEL
LIN {X 0,Y 409.718,Z 1173.532,A -85,B 0,C 180,E1 19170.977,E2 19170.977} C_VEL
LIN {X 0,Y 409.657,Z 1174.188,A -85,B 0,C 180,E1 19168.46,E2 19168.46} C_VEL
LIN {X 0,Y 409.838,Z 1173.061,A -85,B 0,C 180,E1 19165.941,E2 19165.941} C_VEL
LIN {X 0,Y 410.298,Z 1170.122,A -85,B 0,C 180,E1 19163.421,E2 19163.421} C_VEL
LIN {X 0,Y 411.031,Z 1165.485,A -85,B 0,C 180,E1 19161.041,E2 19161.041} C_VEL
LIN {X 0,Y 412.118,Z 1158.942,A -85,B 0,C 180,E1 19158.664,E2 19158.664} C_VEL
LIN {X 0,Y 413.535,Z 1150.736,A -85,B 0,C 180,E1 19156.411,E2 19156.411} C_VEL
LIN {X 0,Y 415.174,Z 1141.084,A -85,B 0,C 180,E1 19154.35,E2 19154.35} C_VEL
LIN {X 0,Y 417.027,Z 1129.748,A -85,B 0,C 180,E1 19152.414,E2 19152.414} C_VEL
LIN {X 0,Y 418.904,Z 1117.399,A -85,B 0,C 180,E1 19150.709,E2 19150.709} C_VEL
LIN {X 0,Y 420.759,Z 1103.773,A -85,B 0,C 180,E1 19149.188,E2 19149.188} C_VEL
LIN {X 0,Y 422.298,Z 1090.589,A -85,B 0,C 180,E1 19147.996,E2 19147.996} C_VEL
LIN {X 0,Y 422.153,Z 1084.005,A -85,B 0,C 180,E1 19147.433,E2 19147.433} C_VEL
LIN {X 0,Y 418.706,Z 1070.198,A -85,B 0,C 180,E1 19146.221,E2 19146.221} C_VEL
LIN {X 0,Y 417.639,Z 1062.318,A -85,B 0,C 180,E1 19145.684,E2 19145.684} C_VEL
LIN {X 0,Y 417.65,Z 1060.252,A -85,B 0,C 180,E1 19145.575,E2 19145.575} C_VEL
LIN {X 0,Y 418.508,Z 1042.961,A -85,B 0,C 180,E1 19144.869,E2 19144.869} C_VEL
LIN {X 0,Y 418.86,Z 1024.848,A -85,B 0,C 180,E1 19144.404,E2 19144.404} C_VEL
LIN {X 0,Y 422.718,Z 866.697,A -85,B 0,C 180,E1 19141.696,E2 19141.696} C_VEL
LIN {X 0,Y 422.181,Z 861.491,A -85,B 0,C 180,E1 19141.532,E2 19141.532} C_VEL
LIN {X 0,Y 425.28,Z 813.289,A -85,B 0,C 180,E1 19137.742,E2 19137.742} C_VEL
LIN {X 0,Y 429.195,Z 763.092,A -85,B 0,C 180,E1 19133.635,E2 19133.635} C_VEL
LIN {X 0,Y 432.981,Z 717.33,A -85,B 0,C 180,E1 19129.853,E2 19129.853} C_VEL
LIN {X 0,Y 433.146,Z 713.88,A -85,B 0,C 180,E1 19129.557,E2 19129.557} C_VEL
LIN {X 0,Y 432.638,Z 711.933,A -85,B 0,C 180,E1 19129.303,E2 19129.303} C_VEL
LIN {X 0,Y 434.56,Z 712.655,A -85,B 0,C 180,E1 19129.021,E2 19129.021} C_VEL
LIN {X 0,Y 437.343,Z 711.783,A -85,B 0,C 180,E1 19128.686,E2 19128.686} C_VEL
LIN {X 0,Y 438.301,Z 711.306,A -85,B 0,C 180,E1 19128.578,E2 19128.578} C_VEL
LIN {X 0,Y 442.353,Z 710.472,A -85,B 0,C 180,E1 19128.09,E2 19128.09} C_VEL
LIN {X 0,Y 446.948,Z 709.484,A -85,B 0,C 180,E1 19127.54,E2 19127.54} C_VEL
LIN {X 0,Y 462.804,Z 732.888,A -85,B 0,C 180,E1 19124.896,E2 19124.896} C_VEL
LIN {X 0,Y 464.638,Z 736.012,A -85,B 0,C 180,E1 19124.595,E2 19124.595} C_VEL
LIN {X 0,Y 444.448,Z 978.632,A -85,B 0,C 180,E1 19119.128,E2 19119.128} C_VEL
LIN {X 0,Y 442.411,Z 1002.045,A -85,B 0,C 180,E1 19118.387,E2 19118.387} C_VEL
LIN {X 0,Y 439.848,Z 1024.473,A -85,B 0,C 180,E1 19117.452,E2 19117.452} C_VEL
LIN {X 0,Y 436.801,Z 1046.085,A -85,B 0,C 180,E1 19116.313,E2 19116.313} C_VEL
LIN {X 0,Y 433.101,Z 1068.516,A -85,B 0,C 180,E1 19114.868,E2 19114.868} C_VEL
LIN {X 0,Y 429.309,Z 1089.15,A -85,B 0,C 180,E1 19113.264,E2 19113.264} C_VEL
LIN {X 0,Y 425.355,Z 1108.634,A -85,B 0,C 180,E1 19111.457,E2 19111.457} C_VEL
LIN {X 0,Y 421.281,Z 1127.245,A -85,B 0,C 180,E1 19109.416,E2 19109.416} C_VEL
LIN {X 0,Y 417.195,Z 1145.257,A -85,B 0,C 180,E1 19107.089,E2 19107.089} C_VEL
LIN {X 0,Y 413.593,Z 1160.909,A -85,B 0,C 180,E1 19104.724,E2 19104.724} C_VEL
LIN {X 0,Y 410.145,Z 1175.828,A -85,B 0,C 180,E1 19102.051,E2 19102.051} C_VEL
LIN {X 0,Y 407.283,Z 1188.602,A -85,B 0,C 180,E1 19099.356,E2 19099.356} C_VEL
LIN {X 0,Y 404.916,Z 1200.11,A -85,B 0,C 180,E1 19096.498,E2 19096.498} C_VEL
LIN {X 0,Y 403.112,Z 1209.695,A -85,B 0,C 180,E1 19093.629,E2 19093.629} C_VEL
LIN {X 0,Y 401.741,Z 1218.371,A -85,B 0,C 180,E1 19090.468,E2 19090.468} C_VEL
LIN {X 0,Y 400.931,Z 1225.024,A -85,B 0,C 180,E1 19087.451,E2 19087.451} C_VEL
LIN {X 0,Y 400.475,Z 1229.985,A -85,B 0,C 180,E1 19084.439,E2 19084.439} C_VEL
LIN {X 0,Y 400.287,Z 1233.713,A -85,B 0,C 180,E1 19081.288,E2 19081.288} C_VEL
LIN {X 0,Y 400.249,Z 1235.703,A -85,B 0,C 180,E1 19078.425,E2 19078.425} C_VEL
LIN {X 0,Y 400.3,Z 1236.48,A -85,B 0,C 180,E1 19075.128,E2 19075.128} C_VEL
LIN {X 0,Y 400.492,Z 1235.787,A -85,B 0,C 180,E1 19072.107,E2 19072.107} C_VEL
LIN {X 0,Y 400.89,Z 1233.501,A -85,B 0,C 180,E1 19068.927,E2 19068.927} C_VEL
LIN {X 0,Y 401.76,Z 1229.397,A -85,B 0,C 180,E1 19065.501,E2 19065.501} C_VEL
LIN {X 0,Y 403.178,Z 1223.836,A -85,B 0,C 180,E1 19062.239,E2 19062.239} C_VEL
LIN {X 0,Y 405.383,Z 1216.238,A -85,B 0,C 180,E1 19058.893,E2 19058.893} C_VEL
LIN {X 0,Y 408.147,Z 1207.475,A -85,B 0,C 180,E1 19055.85,E2 19055.85} C_VEL
LIN {X 0,Y 411.726,Z 1196.873,A -85,B 0,C 180,E1 19052.834,E2 19052.834} C_VEL
LIN {X 0,Y 415.69,Z 1185.493,A -85,B 0,C 180,E1 19050.138,E2 19050.138} C_VEL
LIN {X 0,Y 420.38,Z 1172.075,A -85,B 0,C 180,E1 19047.483,E2 19047.483} C_VEL
LIN {X 0,Y 425.459,Z 1157.103,A -85,B 0,C 180,E1 19045.01,E2 19045.01} C_VEL
LIN {X 0,Y 430.682,Z 1141.004,A -85,B 0,C 180,E1 19042.782,E2 19042.782} C_VEL
LIN {X 0,Y 435.697,Z 1124.578,A -85,B 0,C 180,E1 19040.868,E2 19040.868} C_VEL
LIN {X 0,Y 440.745,Z 1106.791,A -85,B 0,C 180,E1 19039.118,E2 19039.118} C_VEL
LIN {X 0,Y 445.509,Z 1088.396,A -85,B 0,C 180,E1 19037.597,E2 19037.597} C_VEL
LIN {X 0,Y 450.286,Z 1068.053,A -85,B 0,C 180,E1 19036.195,E2 19036.195} C_VEL
LIN {X 0,Y 454.979,Z 1045.905,A -85,B 0,C 180,E1 19034.956,E2 19034.956} C_VEL
LIN {X 0,Y 460.716,Z 1018.994,A -85,B 0,C 180,E1 19033.755,E2 19033.755} C_VEL
LIN {X 0,Y 461.694,Z 1015.253,A -85,B 0,C 180,E1 19033.59,E2 19033.59} C_VEL
LIN {X 0,Y 450.271,Z 1046.651,A -85,B 0,C 180,E1 19031.861,E2 19031.861} C_VEL
LIN {X 0,Y 440.577,Z 1074.871,A -85,B 0,C 180,E1 19029.963,E2 19029.963} C_VEL
LIN {X 0,Y 431.486,Z 1104.159,A -85,B 0,C 180,E1 19027.635,E2 19027.635} C_VEL
LIN {X 0,Y 423.164,Z 1135.747,A -85,B 0,C 180,E1 19024.714,E2 19024.714} C_VEL
LIN {X 0,Y 416.943,Z 1163.545,A -85,B 0,C 180,E1 19021.764,E2 19021.764} C_VEL
LIN {X 0,Y 412.228,Z 1187.288,A -85,B 0,C 180,E1 19018.863,E2 19018.863} C_VEL
LIN {X 0,Y 408.656,Z 1207.219,A -85,B 0,C 180,E1 19016.054,E2 19016.054} C_VEL
LIN {X 0,Y 406.005,Z 1223.672,A -85,B 0,C 180,E1 19013.361,E2 19013.361} C_VEL
LIN {X 0,Y 403.877,Z 1238.167,A -85,B 0,C 180,E1 19010.584,E2 19010.584} C_VEL
LIN {X 0,Y 402.307,Z 1250.324,A -85,B 0,C 180,E1 19007.802,E2 19007.802} C_VEL
LIN {X 0,Y 401.233,Z 1260.36,A -85,B 0,C 180,E1 19005.023,E2 19005.023} C_VEL
LIN {X 0,Y 400.567,Z 1268.826,A -85,B 0,C 180,E1 19002.105,E2 19002.105} C_VEL
LIN {X 0,Y 400.237,Z 1275.069,A -85,B 0,C 180,E1 18999.315,E2 18999.315} C_VEL
LIN {X 0,Y 400.159,Z 1279.685,A -85,B 0,C 180,E1 18996.458,E2 18996.458} C_VEL
LIN {X 0,Y 400.188,Z 1282.441,A -85,B 0,C 180,E1 18993.727,E2 18993.727} C_VEL
LIN {X 0,Y 400.242,Z 1283.607,A -85,B 0,C 180,E1 18991.004,E2 18991.004} C_VEL
LIN {X 0,Y 400.245,Z 1283.242,A -85,B 0,C 180,E1 18988.284,E2 18988.284} C_VEL
LIN {X 0,Y 400.203,Z 1281.234,A -85,B 0,C 180,E1 18985.416,E2 18985.416} C_VEL
LIN {X 0,Y 400.197,Z 1277.583,A -85,B 0,C 180,E1 18982.537,E2 18982.537} C_VEL
LIN {X 0,Y 400.336,Z 1272.258,A -85,B 0,C 180,E1 18979.642,E2 18979.642} C_VEL
LIN {X 0,Y 400.764,Z 1264.796,A -85,B 0,C 180,E1 18976.586,E2 18976.586} C_VEL
LIN {X 0,Y 401.583,Z 1255.915,A -85,B 0,C 180,E1 18973.661,E2 18973.661} C_VEL
LIN {X 0,Y 403.02,Z 1244.268,A -85,B 0,C 180,E1 18970.524,E2 18970.524} C_VEL
LIN {X 0,Y 404.919,Z 1231.61,A -85,B 0,C 180,E1 18967.651,E2 18967.651} C_VEL
LIN {X 0,Y 407.683,Z 1215.672,A -85,B 0,C 180,E1 18964.585,E2 18964.585} C_VEL
LIN {X 0,Y 411.092,Z 1197.943,A -85,B 0,C 180,E1 18961.689,E2 18961.689} C_VEL
LIN {X 0,Y 414.978,Z 1179.241,A -85,B 0,C 180,E1 18959.069,E2 18959.069} C_VEL
LIN {X 0,Y 419.405,Z 1158.667,A -85,B 0,C 180,E1 18956.586,E2 18956.586} C_VEL
LIN {X 0,Y 424.095,Z 1137.349,A -85,B 0,C 180,E1 18954.387,E2 18954.387} C_VEL
LIN {X 0,Y 429.293,Z 1114.079,A -85,B 0,C 180,E1 18952.312,E2 18952.312} C_VEL
LIN {X 0,Y 434.41,Z 1090.871,A -85,B 0,C 180,E1 18950.563,E2 18950.563} C_VEL
LIN {X 0,Y 440.139,Z 1064.291,A -85,B 0,C 180,E1 18948.88,E2 18948.88} C_VEL
LIN {X 0,Y 445.334,Z 1039.209,A -85,B 0,C 180,E1 18947.572,E2 18947.572} C_VEL
LIN {X 0,Y 450.12,Z 1014.009,A -85,B 0,C 180,E1 18946.525,E2 18946.525} C_VEL
LIN {X 0,Y 454.308,Z 987.761,A -85,B 0,C 180,E1 18945.629,E2 18945.629} C_VEL
LIN {X 0,Y 457.425,Z 967.201,A -85,B 0,C 180,E1 18945.122,E2 18945.122} C_VEL
LIN {X 0,Y 458.286,Z 961.507,A -85,B 0,C 180,E1 18945.007,E2 18945.007} C_VEL
LIN {X 0,Y 449.09,Z 939.756,A -85,B 0,C 180,E1 18943.361,E2 18943.361} C_VEL
LIN {X 0,Y 442.142,Z 918.479,A -85,B 0,C 180,E1 18941.894,E2 18941.894} C_VEL
LIN {X 0,Y 441.808,Z 915.849,A -85,B 0,C 180,E1 18941.625,E2 18941.625} C_VEL
LIN {X 0,Y 441.657,Z 893.715,A -85,B 0,C 180,E1 18939.004,E2 18939.004} C_VEL
LIN {X 0,Y 444.155,Z 869.174,A -85,B 0,C 180,E1 18936.303,E2 18936.303} C_VEL
LIN {X 0,Y 451.063,Z 830.848,A -85,B 0,C 180,E1 18932.292,E2 18932.292} C_VEL
LIN {X 0,Y 457.422,Z 797.353,A -85,B 0,C 180,E1 18928.745,E2 18928.745} C_VEL
LIN {X 0,Y 462.391,Z 771.468,A -85,B 0,C 180,E1 18925.97,E2 18925.97} C_VEL
LIN {X 0,Y 456.059,Z 754.754,A -85,B 0,C 180,E1 18922.834,E2 18922.834} C_VEL
LIN {X 0,Y 449.262,Z 737.638,A -85,B 0,C 180,E1 18919.367,E2 18919.367} C_VEL
LIN {X 0,Y 442.574,Z 721.785,A -85,B 0,C 180,E1 18915.865,E2 18915.865} C_VEL
LIN {X 0,Y 436.065,Z 706.877,A -85,B 0,C 180,E1 18912.313,E2 18912.313} C_VEL
LIN {X 0,Y 430.134,Z 693.975,A -85,B 0,C 180,E1 18908.96,E2 18908.96} C_VEL
LIN {X 0,Y 424.851,Z 682.679,A -85,B 0,C 180,E1 18905.808,E2 18905.808} C_VEL
LIN {X 0,Y 419.038,Z 670.45,A -85,B 0,C 180,E1 18902.12,E2 18902.12} C_VEL
LIN {X 0,Y 414.019,Z 660.583,A -85,B 0,C 180,E1 18898.842,E2 18898.842} C_VEL
LIN {X 0,Y 411.614,Z 655.93,A -85,B 0,C 180,E1 18897.215,E2 18897.215} C_VEL
LIN {X 0,Y 409.501,Z 651.603,A -85,B 0,C 180,E1 18895.659,E2 18895.659} C_VEL
LIN {X 0,Y 407.125,Z 646.965,A -85,B 0,C 180,E1 18893.938,E2 18893.938} C_VEL
LIN {X 0,Y 405.297,Z 643.213,A -85,B 0,C 180,E1 18892.487,E2 18892.487} C_VEL
LIN {X 0,Y 402.872,Z 638.91,A -85,B 0,C 180,E1 18890.716,E2 18890.716} C_VEL
LIN {X 0,Y 402.657,Z 637.813,A -85,B 0,C 180,E1 18890.278,E2 18890.278} C_VEL
LIN {X 0,Y 402.668,Z 637.809,A -85,B 0,C 180,E1 18886.355,E2 18886.355} C_VEL
LIN {X 0,Y 402.656,Z 637.817,A -85,B 0,C 180,E1 18882.365,E2 18882.365} C_VEL
LIN {X 0,Y 402.673,Z 637.824,A -85,B 0,C 180,E1 18878.438,E2 18878.438} C_VEL
LIN {X 0,Y 402.664,Z 637.825,A -85,B 0,C 180,E1 18874.336,E2 18874.336} C_VEL
LIN {X 0,Y 402.67,Z 637.819,A -85,B 0,C 180,E1 18870.386,E2 18870.386} C_VEL
LIN {X 0,Y 402.664,Z 637.822,A -85,B 0,C 180,E1 18866.544,E2 18866.544} C_VEL
LIN {X 0,Y 402.664,Z 637.818,A -85,B 0,C 180,E1 18862.527,E2 18862.527} C_VEL
LIN {X 0,Y 402.658,Z 637.798,A -85,B 0,C 180,E1 18858.581,E2 18858.581} C_VEL
LIN {X 0,Y 402.669,Z 637.901,A -85,B 0,C 180,E1 18858.364,E2 18858.364} C_VEL
LIN {X 0,Y 403.947,Z 641.236,A -85,B 0,C 180,E1 18857.87,E2 18857.87} C_VEL
LIN {X 0,Y 404.865,Z 642.786,A -85,B 0,C 180,E1 18857.595,E2 18857.595} C_VEL
LIN {X 0,Y 413.239,Z 660.509,A -85,B 0,C 180,E1 18854.85,E2 18854.85} C_VEL
LIN {X 0,Y 420.793,Z 678.829,A -85,B 0,C 180,E1 18852.254,E2 18852.254} C_VEL
LIN {X 0,Y 427.482,Z 697.898,A -85,B 0,C 180,E1 18849.792,E2 18849.792} C_VEL
LIN {X 0,Y 431.617,Z 712.443,A -85,B 0,C 180,E1 18848.033,E2 18848.033} C_VEL
LIN {X 0,Y 428.227,Z 755.592,A -85,B 0,C 180,E1 18844.488,E2 18844.488} C_VEL
LIN {X 0,Y 424.642,Z 802.466,A -85,B 0,C 180,E1 18840.647,E2 18840.647} C_VEL
LIN {X 0,Y 421.465,Z 851.202,A -85,B 0,C 180,E1 18836.79,E2 18836.79} C_VEL
LIN {X 0,Y 420.974,Z 862.395,A -85,B 0,C 180,E1 18835.964,E2 18835.964} C_VEL
LIN {X 0,Y 421.466,Z 869.576,A -85,B 0,C 180,E1 18835.795,E2 18835.795} C_VEL
LIN {X 0,Y 417.621,Z 1027.972,A -85,B 0,C 180,E1 18833.085,E2 18833.085} C_VEL
LIN {X 0,Y 417.19,Z 1045.682,A -85,B 0,C 180,E1 18832.584,E2 18832.584} C_VEL
LIN {X 0,Y 416.337,Z 1062.664,A -85,B 0,C 180,E1 18831.852,E2 18831.852} C_VEL
LIN {X 0,Y 415.099,Z 1079.06,A -85,B 0,C 180,E1 18830.883,E2 18830.883} C_VEL
LIN {X 0,Y 413.567,Z 1094.254,A -85,B 0,C 180,E1 18829.708,E2 18829.708} C_VEL
LIN {X 0,Y 411.764,Z 1109.165,A -85,B 0,C 180,E1 18828.253,E2 18828.253} C_VEL
LIN {X 0,Y 409.94,Z 1122.356,A -85,B 0,C 180,E1 18826.652,E2 18826.652} C_VEL
LIN {X 0,Y 408.156,Z 1134.021,A -85,B 0,C 180,E1 18824.903,E2 18824.903} C_VEL
LIN {X 0,Y 406.431,Z 1144.63,A -85,B 0,C 180,E1 18822.935,E2 18822.935} C_VEL
LIN {X 0,Y 404.917,Z 1153.786,A -85,B 0,C 180,E1 18820.815,E2 18820.815} C_VEL
LIN {X 0,Y 403.671,Z 1161.479,A -85,B 0,C 180,E1 18818.545,E2 18818.545} C_VEL
LIN {X 0,Y 402.727,Z 1167.545,A -85,B 0,C 180,E1 18816.127,E2 18816.127} C_VEL
LIN {X 0,Y 402.088,Z 1171.957,A -85,B 0,C 180,E1 18813.562,E2 18813.562} C_VEL
LIN {X 0,Y 401.778,Z 1174.492,A -85,B 0,C 180,E1 18810.996,E2 18810.996} C_VEL
LIN {X 0,Y 401.715,Z 1175.139,A -85,B 0,C 180,E1 18808.429,E2 18808.429} C_VEL
LIN {X 0,Y 401.907,Z 1174.005,A -85,B 0,C 180,E1 18805.861,E2 18805.861} C_VEL
LIN {X 0,Y 402.394,Z 1171.057,A -85,B 0,C 180,E1 18803.291,E2 18803.291} C_VEL
LIN {X 0,Y 403.168,Z 1166.41,A -85,B 0,C 180,E1 18800.865,E2 18800.865} C_VEL
LIN {X 0,Y 404.312,Z 1159.858,A -85,B 0,C 180,E1 18798.443,E2 18798.443} C_VEL
LIN {X 0,Y 405.78,Z 1151.731,A -85,B 0,C 180,E1 18796.17,E2 18796.17} C_VEL
LIN {X 0,Y 407.511,Z 1141.972,A -85,B 0,C 180,E1 18794.048,E2 18794.048} C_VEL
LIN {X 0,Y 409.444,Z 1130.622,A -85,B 0,C 180,E1 18792.078,E2 18792.078} C_VEL
LIN {X 0,Y 411.433,Z 1118.035,A -85,B 0,C 180,E1 18790.314,E2 18790.314} C_VEL
LIN {X 0,Y 413.327,Z 1104.597,A -85,B 0,C 180,E1 18788.796,E2 18788.796} C_VEL
LIN {X 0,Y 415.069,Z 1090.041,A -85,B 0,C 180,E1 18787.477,E2 18787.477} C_VEL
LIN {X 0,Y 416.586,Z 1074.545,A -85,B 0,C 180,E1 18786.368,E2 18786.368} C_VEL
LIN {X 0,Y 417.65,Z 1060.252,A -85,B 0,C 180,E1 18785.575,E2 18785.575} C_VEL
LIN {X 0,Y 417.183,Z 1053.034,A -85,B 0,C 180,E1 18785.185,E2 18785.185} C_VEL
LIN {X 0,Y 412.908,Z 1036.911,A -85,B 0,C 180,E1 18784.291,E2 18784.291} C_VEL
LIN {X 0,Y 411.71,Z 1029.492,A -85,B 0,C 180,E1 18784.018,E2 18784.018} C_VEL
LIN {X 0,Y 411.641,Z 1027.306,A -85,B 0,C 180,E1 18783.967,E2 18783.967} C_VEL
LIN {X 0,Y 415.651,Z 867.45,A -85,B 0,C 180,E1 18781.182,E2 18781.182} C_VEL
LIN {X 0,Y 415.123,Z 862.707,A -85,B 0,C 180,E1 18781.042,E2 18781.042} C_VEL
LIN {X 0,Y 418.363,Z 814.601,A -85,B 0,C 180,E1 18777.224,E2 18777.224} C_VEL
LIN {X 0,Y 422.322,Z 765.838,A -85,B 0,C 180,E1 18773.2,E2 18773.2} C_VEL
LIN {X 0,Y 425.899,Z 724.321,A -85,B 0,C 180,E1 18769.742,E2 18769.742} C_VEL
LIN {X 0,Y 427.777,Z 724.772,A -85,B 0,C 180,E1 18769.472,E2 18769.472} C_VEL
LIN {X 0,Y 430.868,Z 723.163,A -85,B 0,C 180,E1 18769.123,E2 18769.123} C_VEL
LIN {X 0,Y 433.761,Z 720.499,A -85,B 0,C 180,E1 18768.841,E2 18768.841} C_VEL
LIN {X 0,Y 437.831,Z 719.418,A -85,B 0,C 180,E1 18768.349,E2 18768.349} C_VEL
LIN {X 0,Y 443.997,Z 717.784,A -85,B 0,C 180,E1 18767.628,E2 18767.628} C_VEL
LIN {X 0,Y 458.408,Z 739.182,A -85,B 0,C 180,E1 18765.196,E2 18765.196} C_VEL
LIN {X 0,Y 437.625,Z 979.313,A -85,B 0,C 180,E1 18759.665,E2 18759.665} C_VEL
LIN {X 0,Y 435.526,Z 1002.775,A -85,B 0,C 180,E1 18758.911,E2 18758.911} C_VEL
LIN {X 0,Y 432.863,Z 1025.344,A -85,B 0,C 180,E1 18757.954,E2 18757.954} C_VEL
LIN {X 0,Y 429.773,Z 1046.659,A -85,B 0,C 180,E1 18756.813,E2 18756.813} C_VEL
LIN {X 0,Y 425.988,Z 1069.051,A -85,B 0,C 180,E1 18755.352,E2 18755.352} C_VEL
LIN {X 0,Y 422.203,Z 1089.199,A -85,B 0,C 180,E1 18753.769,E2 18753.769} C_VEL
LIN {X 0,Y 418.07,Z 1108.989,A -85,B 0,C 180,E1 18751.909,E2 18751.909} C_VEL
LIN {X 0,Y 413.903,Z 1127.564,A -85,B 0,C 180,E1 18749.845,E2 18749.845} C_VEL
LIN {X 0,Y 409.798,Z 1145.207,A -85,B 0,C 180,E1 18747.54,E2 18747.54} C_VEL
LIN {X 0,Y 405.976,Z 1161.365,A -85,B 0,C 180,E1 18745.064,E2 18745.064} C_VEL
LIN {X 0,Y 402.591,Z 1175.552,A -85,B 0,C 180,E1 18742.488,E2 18742.488} C_VEL
LIN {X 0,Y 399.478,Z 1189.106,A -85,B 0,C 180,E1 18739.597,E2 18739.597} C_VEL
LIN {X 0,Y 397.038,Z 1200.638,A -85,B 0,C 180,E1 18736.684,E2 18736.684} C_VEL
LIN {X 0,Y 395.102,Z 1210.683,A -85,B 0,C 180,E1 18733.613,E2 18733.613} C_VEL
LIN {X 0,Y 393.772,Z 1218.923,A -85,B 0,C 180,E1 18730.535,E2 18730.535} C_VEL
LIN {X 0,Y 392.943,Z 1225.581,A -85,B 0,C 180,E1 18727.457,E2 18727.457} C_VEL
LIN {X 0,Y 392.482,Z 1230.544,A -85,B 0,C 180,E1 18724.383,E2 18724.383} C_VEL
LIN {X 0,Y 392.296,Z 1234.27,A -85,B 0,C 180,E1 18721.168,E2 18721.168} C_VEL
LIN {X 0,Y 392.263,Z 1236.265,A -85,B 0,C 180,E1 18718.247,E2 18718.247} C_VEL
LIN {X 0,Y 392.325,Z 1237.046,A -85,B 0,C 180,E1 18715.029,E2 18715.029} C_VEL
LIN {X 0,Y 392.536,Z 1236.401,A -85,B 0,C 180,E1 18711.946,E2 18711.946} C_VEL
LIN {X 0,Y 392.976,Z 1234.199,A -85,B 0,C 180,E1 18708.702,E2 18708.702} C_VEL
LIN {X 0,Y 393.907,Z 1230.287,A -85,B 0,C 180,E1 18705.273,E2 18705.273} C_VEL
LIN {X 0,Y 395.47,Z 1224.729,A -85,B 0,C 180,E1 18701.881,E2 18701.881} C_VEL
LIN {X 0,Y 397.837,Z 1217.227,A -85,B 0,C 180,E1 18698.473,E2 18698.473} C_VEL
LIN {X 0,Y 400.792,Z 1208.6,A -85,B 0,C 180,E1 18695.378,E2 18695.378} C_VEL
LIN {X 0,Y 404.605,Z 1198.163,A -85,B 0,C 180,E1 18692.316,E2 18692.316} C_VEL
LIN {X 0,Y 408.809,Z 1186.969,A -85,B 0,C 180,E1 18689.583,E2 18689.583} C_VEL
LIN {X 0,Y 413.762,Z 1173.778,A -85,B 0,C 180,E1 18686.897,E2 18686.897} C_VEL
LIN {X 0,Y 419.114,Z 1159.08,A -85,B 0,C 180,E1 18684.4,E2 18684.4} C_VEL
LIN {X 0,Y 424.792,Z 1142.889,A -85,B 0,C 180,E1 18682.095,E2 18682.095} C_VEL
LIN {X 0,Y 430.493,Z 1125.663,A -85,B 0,C 180,E1 18680.04,E2 18680.04} C_VEL
LIN {X 0,Y 436.072,Z 1107.58,A -85,B 0,C 180,E1 18678.233,E2 18678.233} C_VEL
LIN {X 0,Y 441.653,Z 1088.045,A -85,B 0,C 180,E1 18676.598,E2 18676.598} C_VEL
LIN {X 0,Y 447.121,Z 1066.99,A -85,B 0,C 180,E1 18675.147,E2 18675.147} C_VEL
LIN {X 0,Y 453.097,Z 1043.061,A -85,B 0,C 180,E1 18673.811,E2 18673.811} C_VEL
LIN {X 0,Y 454.521,Z 1037.295,A -85,B 0,C 180,E1 18673.518,E2 18673.518} C_VEL
LIN {X 0,Y 444.043,Z 1062.365,A -85,B 0,C 180,E1 18671.975,E2 18671.975} C_VEL
LIN {X 0,Y 433.702,Z 1088.38,A -85,B 0,C 180,E1 18670.035,E2 18670.035} C_VEL
LIN {X 0,Y 424.105,Z 1115.567,A -85,B 0,C 180,E1 18667.637,E2 18667.637} C_VEL
LIN {X 0,Y 415.227,Z 1145.951,A -85,B 0,C 180,E1 18664.557,E2 18664.557} C_VEL
LIN {X 0,Y 408.595,Z 1172.912,A -85,B 0,C 180,E1 18661.417,E2 18661.417} C_VEL
LIN {X 0,Y 403.654,Z 1196.061,A -85,B 0,C 180,E1 18658.32,E2 18658.32} C_VEL
LIN {X 0,Y 400.15,Z 1214.546,A -85,B 0,C 180,E1 18655.456,E2 18655.456} C_VEL
LIN {X 0,Y 397.391,Z 1230.516,A -85,B 0,C 180,E1 18652.568,E2 18652.568} C_VEL
LIN {X 0,Y 395.431,Z 1243.45,A -85,B 0,C 180,E1 18649.808,E2 18649.808} C_VEL
LIN {X 0,Y 393.957,Z 1254.586,A -85,B 0,C 180,E1 18646.972,E2 18646.972} C_VEL
LIN {X 0,Y 392.99,Z 1263.72,A -85,B 0,C 180,E1 18644.14,E2 18644.14} C_VEL
LIN {X 0,Y 392.418,Z 1271.299,A -85,B 0,C 180,E1 18641.168,E2 18641.168} C_VEL
LIN {X 0,Y 392.2,Z 1276.701,A -85,B 0,C 180,E1 18638.358,E2 18638.358} C_VEL
LIN {X 0,Y 392.168,Z 1280.437,A -85,B 0,C 180,E1 18635.562,E2 18635.562} C_VEL
LIN {X 0,Y 392.22,Z 1282.572,A -85,B 0,C 180,E1 18632.778,E2 18632.778} C_VEL
LIN {X 0,Y 392.282,Z 1283.114,A -85,B 0,C 180,E1 18630.002,E2 18630.002} C_VEL
LIN {X 0,Y 392.251,Z 1282.012,A -85,B 0,C 180,E1 18627.08,E2 18627.08} C_VEL
LIN {X 0,Y 392.214,Z 1279.249,A -85,B 0,C 180,E1 18624.149,E2 18624.149} C_VEL
LIN {X 0,Y 392.247,Z 1274.831,A -85,B 0,C 180,E1 18621.204,E2 18621.204} C_VEL
LIN {X 0,Y 392.496,Z 1268.701,A -85,B 0,C 180,E1 18618.243,E2 18618.243} C_VEL
LIN {X 0,Y 393.123,Z 1260.36,A -85,B 0,C 180,E1 18615.117,E2 18615.117} C_VEL
LIN {X 0,Y 394.185,Z 1250.575,A -85,B 0,C 180,E1 18612.128,E2 18612.128} C_VEL
LIN {X 0,Y 395.919,Z 1238.156,A -85,B 0,C 180,E1 18608.987,E2 18608.987} C_VEL
LIN {X 0,Y 398.246,Z 1224.196,A -85,B 0,C 180,E1 18606.002,E2 18606.002} C_VEL
LIN {X 0,Y 401.303,Z 1207.932,A -85,B 0,C 180,E1 18603.036,E2 18603.036} C_VEL
LIN {X 0,Y 405.181,Z 1189.038,A -85,B 0,C 180,E1 18600.103,E2 18600.103} C_VEL
LIN {X 0,Y 409.509,Z 1169.158,A -85,B 0,C 180,E1 18597.464,E2 18597.464} C_VEL
LIN {X 0,Y 414.157,Z 1148.475,A -85,B 0,C 180,E1 18595.1,E2 18595.1} C_VEL
LIN {X 0,Y 419.778,Z 1123.834,A -85,B 0,C 180,E1 18592.71,E2 18592.71} C_VEL
LIN {X 0,Y 424.979,Z 1101.134,A -85,B 0,C 180,E1 18590.825,E2 18590.825} C_VEL
LIN {X 0,Y 430.337,Z 1077.247,A -85,B 0,C 180,E1 18589.154,E2 18589.154} C_VEL
LIN {X 0,Y 435.747,Z 1052.715,A -85,B 0,C 180,E1 18587.705,E2 18587.705} C_VEL
LIN {X 0,Y 440.874,Z 1027.64,A -85,B 0,C 180,E1 18586.505,E2 18586.505} C_VEL
LIN {X 0,Y 445.891,Z 1000.297,A -85,B 0,C 180,E1 18585.447,E2 18585.447} C_VEL
LIN {X 0,Y 449.482,Z 976.818,A -85,B 0,C 180,E1 18584.725,E2 18584.725} C_VEL
LIN {X 0,Y 451.527,Z 963.824,A -85,B 0,C 180,E1 18584.433,E2 18584.433} C_VEL
LIN {X 0,Y 443.174,Z 943.67,A -85,B 0,C 180,E1 18582.885,E2 18582.885} C_VEL
LIN {X 0,Y 436.278,Z 922.157,A -85,B 0,C 180,E1 18581.37,E2 18581.37} C_VEL
LIN {X 0,Y 434.485,Z 915.196,A -85,B 0,C 180,E1 18580.899,E2 18580.899} C_VEL
LIN {X 0,Y 434.796,Z 892.495,A -85,B 0,C 180,E1 18578.215,E2 18578.215} C_VEL
LIN {X 0,Y 437.821,Z 867.845,A -85,B 0,C 180,E1 18575.488,E2 18575.488} C_VEL
LIN {X 0,Y 444.761,Z 830.724,A -85,B 0,C 180,E1 18571.569,E2 18571.569} C_VEL
LIN {X 0,Y 451.254,Z 797.489,A -85,B 0,C 180,E1 18568.018,E2 18568.018} C_VEL
LIN {X 0,Y 455.651,Z 774.865,A -85,B 0,C 180,E1 18565.544,E2 18565.544} C_VEL
LIN {X 0,Y 448.72,Z 756.537,A -85,B 0,C 180,E1 18562.038,E2 18562.038} C_VEL
LIN {X 0,Y 441.591,Z 738.741,A -85,B 0,C 180,E1 18558.345,E2 18558.345} C_VEL
LIN {X 0,Y 435.167,Z 723.573,A -85,B 0,C 180,E1 18554.913,E2 18554.913} C_VEL
LIN {X 0,Y 428.953,Z 709.338,A -85,B 0,C 180,E1 18551.428,E2 18551.428} C_VEL
LIN {X 0,Y 423.038,Z 696.46,A -85,B 0,C 180,E1 18547.987,E2 18547.987} C_VEL
LIN {X 0,Y 417.476,Z 684.442,A -85,B 0,C 180,E1 18544.533,E2 18544.533} C_VEL
LIN {X 0,Y 412.28,Z 674.036,A -85,B 0,C 180,E1 18541.251,E2 18541.251} C_VEL
LIN {X 0,Y 408.393,Z 666.073,A -85,B 0,C 180,E1 18538.597,E2 18538.597} C_VEL
LIN {X 0,Y 406.096,Z 661.6,A -85,B 0,C 180,E1 18537.036,E2 18537.036} C_VEL
LIN {X 0,Y 403.976,Z 657.267,A -85,B 0,C 180,E1 18535.457,E2 18535.457} C_VEL
LIN {X 0,Y 401.584,Z 652.624,A -85,B 0,C 180,E1 18533.71,E2 18533.71} C_VEL
LIN {X 0,Y 399.315,Z 648.092,A -85,B 0,C 180,E1 18531.939,E2 18531.939} C_VEL
LIN {X 0,Y 397.416,Z 644.439,A -85,B 0,C 180,E1 18530.441,E2 18530.441} C_VEL
LIN {X 0,Y 396.646,Z 643.087,A -85,B 0,C 180,E1 18529.836,E2 18529.836} C_VEL
LIN {X 0,Y 394.916,Z 639.848,A -85,B 0,C 180,E1 18528.462,E2 18528.462} C_VEL
LIN {X 0,Y 394.726,Z 638.813,A -85,B 0,C 180,E1 18528.011,E2 18528.011} C_VEL
LIN {X 0,Y 394.721,Z 638.803,A -85,B 0,C 180,E1 18524.122,E2 18524.122} C_VEL
LIN {X 0,Y 394.725,Z 638.799,A -85,B 0,C 180,E1 18520.157,E2 18520.157} C_VEL
LIN {X 0,Y 394.719,Z 638.798,A -85,B 0,C 180,E1 18516.248,E2 18516.248} C_VEL
LIN {X 0,Y 394.735,Z 638.796,A -85,B 0,C 180,E1 18512.219,E2 18512.219} C_VEL
LIN {X 0,Y 394.727,Z 638.799,A -85,B 0,C 180,E1 18508.204,E2 18508.204} C_VEL
LIN {X 0,Y 394.72,Z 638.799,A -85,B 0,C 180,E1 18504.185,E2 18504.185} C_VEL
LIN {X 0,Y 394.728,Z 638.803,A -85,B 0,C 180,E1 18500.331,E2 18500.331} C_VEL
LIN {X 0,Y 394.744,Z 638.896,A -85,B 0,C 180,E1 18499.384,E2 18499.384} C_VEL
LIN {X 0,Y 395.805,Z 641.91,A -85,B 0,C 180,E1 18498.942,E2 18498.942} C_VEL
LIN {X 0,Y 397.117,Z 644.171,A -85,B 0,C 180,E1 18498.532,E2 18498.532} C_VEL
LIN {X 0,Y 404.629,Z 659.578,A -85,B 0,C 180,E1 18496.021,E2 18496.021} C_VEL
LIN {X 0,Y 411.92,Z 676.693,A -85,B 0,C 180,E1 18493.465,E2 18493.465} C_VEL
LIN {X 0,Y 418.887,Z 695.489,A -85,B 0,C 180,E1 18490.931,E2 18490.931} C_VEL
LIN {X 0,Y 424.819,Z 714.95,A -85,B 0,C 180,E1 18488.508,E2 18488.508} C_VEL
LIN {X 0,Y 421.366,Z 756.455,A -85,B 0,C 180,E1 18485.045,E2 18485.045} C_VEL
LIN {X 0,Y 417.644,Z 803.905,A -85,B 0,C 180,E1 18481.137,E2 18481.137} C_VEL
LIN {X 0,Y 414.435,Z 851.131,A -85,B 0,C 180,E1 18477.367,E2 18477.367} C_VEL
LIN {X 0,Y 413.855,Z 863.291,A -85,B 0,C 180,E1 18476.457,E2 18476.457} C_VEL
LIN {X 0,Y 414.334,Z 870.468,A -85,B 0,C 180,E1 18476.285,E2 18476.285} C_VEL
LIN {X 0,Y 410.346,Z 1028.488,A -85,B 0,C 180,E1 18473.54,E2 18473.54} C_VEL
LIN {X 0,Y 409.905,Z 1046.184,A -85,B 0,C 180,E1 18473.037,E2 18473.037} C_VEL
LIN {X 0,Y 409.03,Z 1063.12,A -85,B 0,C 180,E1 18472.301,E2 18472.301} C_VEL
LIN {X 0,Y 407.791,Z 1079.124,A -85,B 0,C 180,E1 18471.351,E2 18471.351} C_VEL
LIN {X 0,Y 406.205,Z 1094.541,A -85,B 0,C 180,E1 18470.156,E2 18470.156} C_VEL
LIN {X 0,Y 404.408,Z 1108.952,A -85,B 0,C 180,E1 18468.744,E2 18468.744} C_VEL
LIN {X 0,Y 402.501,Z 1122.32,A -85,B 0,C 180,E1 18467.118,E2 18467.118} C_VEL
LIN {X 0,Y 400.634,Z 1134.204,A -85,B 0,C 180,E1 18465.338,E2 18465.338} C_VEL
LIN {X 0,Y 398.817,Z 1144.961,A -85,B 0,C 180,E1 18463.334,E2 18463.334} C_VEL
LIN {X 0,Y 397.12,Z 1154.783,A -85,B 0,C 180,E1 18461.03,E2 18461.03} C_VEL
LIN {X 0,Y 395.819,Z 1162.467,A -85,B 0,C 180,E1 18458.716,E2 18458.716} C_VEL
LIN {X 0,Y 394.831,Z 1168.522,A -85,B 0,C 180,E1 18456.25,E2 18456.25} C_VEL
LIN {X 0,Y 394.162,Z 1172.927,A -85,B 0,C 180,E1 18453.634,E2 18453.634} C_VEL
LIN {X 0,Y 393.837,Z 1175.452,A -85,B 0,C 180,E1 18451.016,E2 18451.016} C_VEL
LIN {X 0,Y 393.773,Z 1176.09,A -85,B 0,C 180,E1 18448.397,E2 18448.397} C_VEL
LIN {X 0,Y 393.978,Z 1174.949,A -85,B 0,C 180,E1 18445.777,E2 18445.777} C_VEL
LIN {X 0,Y 394.493,Z 1171.993,A -85,B 0,C 180,E1 18443.156,E2 18443.156} C_VEL
LIN {X 0,Y 395.309,Z 1167.335,A -85,B 0,C 180,E1 18440.682,E2 18440.682} C_VEL
LIN {X 0,Y 396.513,Z 1160.774,A -85,B 0,C 180,E1 18438.212,E2 18438.212} C_VEL
LIN {X 0,Y 398.052,Z 1152.637,A -85,B 0,C 180,E1 18435.896,E2 18435.896} C_VEL
LIN {X 0,Y 399.86,Z 1142.861,A -85,B 0,C 180,E1 18433.734,E2 18433.734} C_VEL
LIN {X 0,Y 401.876,Z 1131.496,A -85,B 0,C 180,E1 18431.728,E2 18431.728} C_VEL
LIN {X 0,Y 403.929,Z 1119.002,A -85,B 0,C 180,E1 18429.948,E2 18429.948} C_VEL
LIN {X 0,Y 405.889,Z 1105.624,A -85,B 0,C 180,E1 18428.41,E2 18428.41} C_VEL
LIN {X 0,Y 407.725,Z 1090.834,A -85,B 0,C 180,E1 18427.048,E2 18427.048} C_VEL
LIN {X 0,Y 409.302,Z 1075.295,A -85,B 0,C 180,E1 18425.921,E2 18425.921} C_VEL
LIN {X 0,Y 410.563,Z 1058.68,A -85,B 0,C 180,E1 18425.003,E2 18425.003} C_VEL
LIN {X 0,Y 411.351,Z 1041.474,A -85,B 0,C 180,E1 18424.334,E2 18424.334} C_VEL
LIN {X 0,Y 411.641,Z 1027.306,A -85,B 0,C 180,E1 18423.967,E2 18423.967} C_VEL
LIN {X 0,Y 410.817,Z 1019.724,A -85,B 0,C 180,E1 18423.76,E2 18423.76} C_VEL
LIN {X 0,Y 405.65,Z 999.844,A -85,B 0,C 180,E1 18423.013,E2 18423.013} C_VEL
LIN {X 0,Y 405.161,Z 993.318,A -85,B 0,C 180,E1 18422.85,E2 18422.85} C_VEL
LIN {X 0,Y 408.643,Z 868.41,A -85,B 0,C 180,E1 18420.656,E2 18420.656} C_VEL
LIN {X 0,Y 408.13,Z 863.448,A -85,B 0,C 180,E1 18420.497,E2 18420.497} C_VEL
LIN {X 0,Y 411.542,Z 814.893,A -85,B 0,C 180,E1 18416.61,E2 18416.61} C_VEL
LIN {X 0,Y 415.672,Z 765.561,A -85,B 0,C 180,E1 18412.511,E2 18412.511} C_VEL
LIN {X 0,Y 418.178,Z 738.739,A -85,B 0,C 180,E1 18410.236,E2 18410.236} C_VEL
LIN {X 0,Y 419.892,Z 739.137,A -85,B 0,C 180,E1 18409.986,E2 18409.986} C_VEL
LIN {X 0,Y 422.974,Z 737.548,A -85,B 0,C 180,E1 18409.628,E2 18409.628} C_VEL
LIN {X 0,Y 427.141,Z 733.076,A -85,B 0,C 180,E1 18409.244,E2 18409.244} C_VEL
LIN {X 0,Y 427.674,Z 732.5,A -85,B 0,C 180,E1 18409.195,E2 18409.195} C_VEL
LIN {X 0,Y 431.697,Z 730.734,A -85,B 0,C 180,E1 18408.734,E2 18408.734} C_VEL
LIN {X 0,Y 435.135,Z 728.053,A -85,B 0,C 180,E1 18408.386,E2 18408.386} C_VEL
LIN {X 0,Y 441.229,Z 726.342,A -85,B 0,C 180,E1 18407.674,E2 18407.674} C_VEL
LIN {X 0,Y 452.16,Z 742.855,A -85,B 0,C 180,E1 18405.794,E2 18405.794} C_VEL
LIN {X 0,Y 430.86,Z 979.369,A -85,B 0,C 180,E1 18400.23,E2 18400.23} C_VEL
LIN {X 0,Y 428.739,Z 1002.62,A -85,B 0,C 180,E1 18399.478,E2 18399.478} C_VEL
LIN {X 0,Y 425.963,Z 1025.483,A -85,B 0,C 180,E1 18398.496,E2 18398.496} C_VEL
LIN {X 0,Y 422.807,Z 1046.839,A -85,B 0,C 180,E1 18397.344,E2 18397.344} C_VEL
LIN {X 0,Y 419.113,Z 1068.289,A -85,B 0,C 180,E1 18395.937,E2 18395.937} C_VEL
LIN {X 0,Y 415.105,Z 1089.14,A -85,B 0,C 180,E1 18394.287,E2 18394.287} C_VEL
LIN {X 0,Y 410.95,Z 1108.538,A -85,B 0,C 180,E1 18392.446,E2 18392.446} C_VEL
LIN {X 0,Y 406.525,Z 1127.872,A -85,B 0,C 180,E1 18390.28,E2 18390.28} C_VEL
LIN {X 0,Y 402.423,Z 1145.083,A -85,B 0,C 180,E1 18388.009,E2 18388.009} C_VEL
LIN {X 0,Y 398.578,Z 1160.863,A -85,B 0,C 180,E1 18385.562,E2 18385.562} C_VEL
LIN {X 0,Y 395.057,Z 1175.239,A -85,B 0,C 180,E1 18382.941,E2 18382.941} C_VEL
LIN {X 0,Y 391.823,Z 1188.958,A -85,B 0,C 180,E1 18379.996,E2 18379.996} C_VEL
LIN {X 0,Y 389.276,Z 1200.619,A -85,B 0,C 180,E1 18377.027,E2 18377.027} C_VEL
LIN {X 0,Y 387.228,Z 1210.874,A -85,B 0,C 180,E1 18373.852,E2 18373.852} C_VEL
LIN {X 0,Y 385.803,Z 1219.455,A -85,B 0,C 180,E1 18370.604,E2 18370.604} C_VEL
LIN {X 0,Y 384.953,Z 1226.123,A -85,B 0,C 180,E1 18367.462,E2 18367.462} C_VEL
LIN {X 0,Y 384.488,Z 1231.093,A -85,B 0,C 180,E1 18364.325,E2 18364.325} C_VEL
LIN {X 0,Y 384.305,Z 1234.823,A -85,B 0,C 180,E1 18361.044,E2 18361.044} C_VEL
LIN {X 0,Y 384.277,Z 1236.825,A -85,B 0,C 180,E1 18358.062,E2 18358.062} C_VEL
LIN {X 0,Y 384.359,Z 1237.609,A -85,B 0,C 180,E1 18354.776,E2 18354.776} C_VEL
LIN {X 0,Y 384.612,Z 1236.932,A -85,B 0,C 180,E1 18351.478,E2 18351.478} C_VEL
LIN {X 0,Y 385.132,Z 1234.658,A -85,B 0,C 180,E1 18348.164,E2 18348.164} C_VEL
LIN {X 0,Y 386.197,Z 1230.71,A -85,B 0,C 180,E1 18344.687,E2 18344.687} C_VEL
LIN {X 0,Y 387.87,Z 1225.363,A -85,B 0,C 180,E1 18341.358,E2 18341.358} C_VEL
LIN {X 0,Y 390.458,Z 1217.923,A -85,B 0,C 180,E1 18337.887,E2 18337.887} C_VEL
LIN {X 0,Y 393.684,Z 1209.279,A -85,B 0,C 180,E1 18334.716,E2 18334.716} C_VEL
LIN {X 0,Y 397.967,Z 1198.456,A -85,B 0,C 180,E1 18331.486,E2 18331.486} C_VEL
LIN {X 0,Y 403.014,Z 1185.932,A -85,B 0,C 180,E1 18328.433,E2 18328.433} C_VEL
LIN {X 0,Y 408.393,Z 1172.552,A -85,B 0,C 180,E1 18325.728,E2 18325.728} C_VEL
LIN {X 0,Y 414.029,Z 1158.25,A -85,B 0,C 180,E1 18323.303,E2 18323.303} C_VEL
LIN {X 0,Y 420.172,Z 1141.95,A -85,B 0,C 180,E1 18320.991,E2 18320.991} C_VEL
LIN {X 0,Y 426.286,Z 1124.756,A -85,B 0,C 180,E1 18318.946,E2 18318.946} C_VEL
LIN {X 0,Y 432.28,Z 1106.779,A -85,B 0,C 180,E1 18317.153,E2 18317.153} C_VEL
LIN {X 0,Y 438.784,Z 1085.949,A -85,B 0,C 180,E1 18315.423,E2 18315.423} C_VEL
LIN {X 0,Y 445.473,Z 1063.631,A -85,B 0,C 180,E1 18313.904,E2 18313.904} C_VEL
LIN {X 0,Y 447.497,Z 1056.864,A -85,B 0,C 180,E1 18313.489,E2 18313.489} C_VEL
LIN {X 0,Y 435.829,Z 1080.883,A -85,B 0,C 180,E1 18311.797,E2 18311.797} C_VEL
LIN {X 0,Y 424.885,Z 1105.331,A -85,B 0,C 180,E1 18309.713,E2 18309.713} C_VEL
LIN {X 0,Y 414.557,Z 1132.475,A -85,B 0,C 180,E1 18306.999,E2 18306.999} C_VEL
LIN {X 0,Y 405.256,Z 1162.589,A -85,B 0,C 180,E1 18303.553,E2 18303.553} C_VEL
LIN {X 0,Y 398.842,Z 1187.593,A -85,B 0,C 180,E1 18300.26,E2 18300.26} C_VEL
LIN {X 0,Y 394.282,Z 1207.969,A -85,B 0,C 180,E1 18297.162,E2 18297.162} C_VEL
LIN {X 0,Y 390.92,Z 1224.957,A -85,B 0,C 180,E1 18294.159,E2 18294.159} C_VEL
LIN {X 0,Y 388.463,Z 1238.861,A -85,B 0,C 180,E1 18291.282,E2 18291.282} C_VEL
LIN {X 0,Y 386.63,Z 1250.79,A -85,B 0,C 180,E1 18288.354,E2 18288.354} C_VEL
LIN {X 0,Y 385.361,Z 1260.888,A -85,B 0,C 180,E1 18285.348,E2 18285.348} C_VEL
LIN {X 0,Y 384.605,Z 1268.971,A -85,B 0,C 180,E1 18282.311,E2 18282.311} C_VEL
LIN {X 0,Y 384.246,Z 1274.835,A -85,B 0,C 180,E1 18279.438,E2 18279.438} C_VEL
LIN {X 0,Y 384.166,Z 1279.01,A -85,B 0,C 180,E1 18276.578,E2 18276.578} C_VEL
LIN {X 0,Y 384.211,Z 1281.563,A -85,B 0,C 180,E1 18273.732,E2 18273.732} C_VEL
LIN {X 0,Y 384.278,Z 1282.542,A -85,B 0,C 180,E1 18270.897,E2 18270.897} C_VEL
LIN {X 0,Y 384.287,Z 1281.968,A -85,B 0,C 180,E1 18268.064,E2 18268.064} C_VEL
LIN {X 0,Y 384.247,Z 1279.722,A -85,B 0,C 180,E1 18265.076,E2 18265.076} C_VEL
LIN {X 0,Y 384.235,Z 1275.763,A -85,B 0,C 180,E1 18262.075,E2 18262.075} C_VEL
LIN {X 0,Y 384.415,Z 1270.09,A -85,B 0,C 180,E1 18259.057,E2 18259.057} C_VEL
LIN {X 0,Y 384.934,Z 1262.293,A -85,B 0,C 180,E1 18255.869,E2 18255.869} C_VEL
LIN {X 0,Y 385.883,Z 1252.961,A -85,B 0,C 180,E1 18252.821,E2 18252.821} C_VEL
LIN {X 0,Y 387.493,Z 1241.137,A -85,B 0,C 180,E1 18249.616,E2 18249.616} C_VEL
LIN {X 0,Y 389.822,Z 1226.988,A -85,B 0,C 180,E1 18246.416,E2 18246.416} C_VEL
LIN {X 0,Y 392.631,Z 1212.057,A -85,B 0,C 180,E1 18243.537,E2 18243.537} C_VEL
LIN {X 0,Y 396.393,Z 1193.904,A -85,B 0,C 180,E1 18240.538,E2 18240.538} C_VEL
LIN {X 0,Y 401.039,Z 1172.869,A -85,B 0,C 180,E1 18237.588,E2 18237.588} C_VEL
LIN {X 0,Y 406.361,Z 1149.79,A -85,B 0,C 180,E1 18234.849,E2 18234.849} C_VEL
LIN {X 0,Y 412.105,Z 1125.27,A -85,B 0,C 180,E1 18232.398,E2 18232.398} C_VEL
LIN {X 0,Y 417.407,Z 1102.671,A -85,B 0,C 180,E1 18230.475,E2 18230.475} C_VEL
LIN {X 0,Y 423.415,Z 1076.738,A -85,B 0,C 180,E1 18228.61,E2 18228.61} C_VEL
LIN {X 0,Y 429.041,Z 1051.879,A -85,B 0,C 180,E1 18227.12,E2 18227.12} C_VEL
LIN {X 0,Y 434.425,Z 1026.222,A -85,B 0,C 180,E1 18225.877,E2 18225.877} C_VEL
LIN {X 0,Y 439.548,Z 999.021,A -85,B 0,C 180,E1 18224.809,E2 18224.809} C_VEL
LIN {X 0,Y 443.119,Z 976.478,A -85,B 0,C 180,E1 18224.103,E2 18224.103} C_VEL
LIN {X 0,Y 444.711,Z 966.15,A -85,B 0,C 180,E1 18223.843,E2 18223.843} C_VEL
LIN {X 0,Y 436.533,Z 945.323,A -85,B 0,C 180,E1 18222.232,E2 18222.232} C_VEL
LIN {X 0,Y 430.236,Z 925.331,A -85,B 0,C 180,E1 18220.817,E2 18220.817} C_VEL
LIN {X 0,Y 427.197,Z 912.984,A -85,B 0,C 180,E1 18219.978,E2 18219.978} C_VEL
LIN {X 0,Y 428.2,Z 889.615,A -85,B 0,C 180,E1 18217.214,E2 18217.214} C_VEL
LIN {X 0,Y 432.148,Z 863.188,A -85,B 0,C 180,E1 18214.313,E2 18214.313} C_VEL
LIN {X 0,Y 439.105,Z 827.7,A -85,B 0,C 180,E1 18210.517,E2 18210.517} C_VEL
LIN {X 0,Y 445.974,Z 793.66,A -85,B 0,C 180,E1 18206.838,E2 18206.838} C_VEL
LIN {X 0,Y 448.983,Z 778.578,A -85,B 0,C 180,E1 18205.174,E2 18205.174} C_VEL
LIN {X 0,Y 442.148,Z 760.412,A -85,B 0,C 180,E1 18201.658,E2 18201.658} C_VEL
LIN {X 0,Y 435.585,Z 743.906,A -85,B 0,C 180,E1 18198.191,E2 18198.191} C_VEL
LIN {X 0,Y 429.184,Z 728.666,A -85,B 0,C 180,E1 18194.711,E2 18194.711} C_VEL
LIN {X 0,Y 422.712,Z 713.741,A -85,B 0,C 180,E1 18191.008,E2 18191.008} C_VEL
LIN {X 0,Y 416.91,Z 701.108,A -85,B 0,C 180,E1 18187.58,E2 18187.58} C_VEL
LIN {X 0,Y 411.731,Z 689.822,A -85,B 0,C 180,E1 18184.318,E2 18184.318} C_VEL
LIN {X 0,Y 406.536,Z 679.319,A -85,B 0,C 180,E1 18180.986,E2 18180.986} C_VEL
LIN {X 0,Y 402.86,Z 671.741,A -85,B 0,C 180,E1 18178.436,E2 18178.436} C_VEL
LIN {X 0,Y 400.367,Z 666.9,A -85,B 0,C 180,E1 18176.707,E2 18176.707} C_VEL
LIN {X 0,Y 398.336,Z 662.764,A -85,B 0,C 180,E1 18175.196,E2 18175.196} C_VEL
LIN {X 0,Y 396.053,Z 658.262,A -85,B 0,C 180,E1 18173.477,E2 18173.477} C_VEL
LIN {X 0,Y 393.727,Z 653.705,A -85,B 0,C 180,E1 18171.677,E2 18171.677} C_VEL
LIN {X 0,Y 391.557,Z 649.277,A -85,B 0,C 180,E1 18169.851,E2 18169.851} C_VEL
LIN {X 0,Y 389.58,Z 645.738,A -85,B 0,C 180,E1 18168.301,E2 18168.301} C_VEL
LIN {X 0,Y 388.899,Z 644.286,A -85,B 0,C 180,E1 18167.677,E2 18167.677} C_VEL
LIN {X 0,Y 387.005,Z 640.865,A -85,B 0,C 180,E1 18166.097,E2 18166.097} C_VEL
LIN {X 0,Y 386.778,Z 639.794,A -85,B 0,C 180,E1 18165.63,E2 18165.63} C_VEL
LIN {X 0,Y 386.792,Z 639.804,A -85,B 0,C 180,E1 18161.564,E2 18161.564} C_VEL
LIN {X 0,Y 386.788,Z 639.794,A -85,B 0,C 180,E1 18157.505,E2 18157.505} C_VEL
LIN {X 0,Y 386.783,Z 639.787,A -85,B 0,C 180,E1 18153.433,E2 18153.433} C_VEL
LIN {X 0,Y 386.79,Z 639.784,A -85,B 0,C 180,E1 18149.385,E2 18149.385} C_VEL
LIN {X 0,Y 386.785,Z 639.782,A -85,B 0,C 180,E1 18145.288,E2 18145.288} C_VEL
LIN {X 0,Y 386.782,Z 639.785,A -85,B 0,C 180,E1 18141.273,E2 18141.273} C_VEL
LIN {X 0,Y 386.812,Z 639.943,A -85,B 0,C 180,E1 18140.478,E2 18140.478} C_VEL
LIN {X 0,Y 388.199,Z 643.426,A -85,B 0,C 180,E1 18139.914,E2 18139.914} C_VEL
LIN {X 0,Y 389.28,Z 645.228,A -85,B 0,C 180,E1 18139.566,E2 18139.566} C_VEL
LIN {X 0,Y 397.047,Z 660.888,A -85,B 0,C 180,E1 18136.909,E2 18136.909} C_VEL
LIN {X 0,Y 405.015,Z 679.285,A -85,B 0,C 180,E1 18134.076,E2 18134.076} C_VEL
LIN {X 0,Y 412.074,Z 698.39,A -85,B 0,C 180,E1 18131.428,E2 18131.428} C_VEL
LIN {X 0,Y 417.923,Z 717.711,A -85,B 0,C 180,E1 18128.961,E2 18128.961} C_VEL
LIN {X 0,Y 414.762,Z 755.724,A -85,B 0,C 180,E1 18125.772,E2 18125.772} C_VEL
LIN {X 0,Y 410.842,Z 803.491,A -85,B 0,C 180,E1 18121.802,E2 18121.802} C_VEL
LIN {X 0,Y 407.368,Z 852.026,A -85,B 0,C 180,E1 18117.883,E2 18117.883} C_VEL
LIN {X 0,Y 406.766,Z 864.171,A -85,B 0,C 180,E1 18116.968,E2 18116.968} C_VEL
LIN {X 0,Y 407.231,Z 871.353,A -85,B 0,C 180,E1 18116.791,E2 18116.791} C_VEL
LIN {X 0,Y 403.096,Z 1028.836,A -85,B 0,C 180,E1 18114.014,E2 18114.014} C_VEL
LIN {X 0,Y 402.656,Z 1046.444,A -85,B 0,C 180,E1 18113.515,E2 18113.515} C_VEL
LIN {X 0,Y 401.731,Z 1063.861,A -85,B 0,C 180,E1 18112.752,E2 18112.752} C_VEL
LIN {X 0,Y 400.407,Z 1080.344,A -85,B 0,C 180,E1 18111.757,E2 18111.757} C_VEL
LIN {X 0,Y 398.769,Z 1095.61,A -85,B 0,C 180,E1 18110.549,E2 18110.549} C_VEL
LIN {X 0,Y 396.819,Z 1110.621,A -85,B 0,C 180,E1 18109.043,E2 18109.043} C_VEL
LIN {X 0,Y 394.846,Z 1123.89,A -85,B 0,C 180,E1 18107.384,E2 18107.384} C_VEL
LIN {X 0,Y 392.839,Z 1136.053,A -85,B 0,C 180,E1 18105.499,E2 18105.499} C_VEL
LIN {X 0,Y 390.973,Z 1146.642,A -85,B 0,C 180,E1 18103.455,E2 18103.455} C_VEL
LIN {X 0,Y 389.329,Z 1155.78,A -85,B 0,C 180,E1 18101.253,E2 18101.253} C_VEL
LIN {X 0,Y 387.971,Z 1163.455,A -85,B 0,C 180,E1 18098.893,E2 18098.893} C_VEL
LIN {X 0,Y 386.936,Z 1169.499,A -85,B 0,C 180,E1 18096.378,E2 18096.378} C_VEL
LIN {X 0,Y 386.237,Z 1173.896,A -85,B 0,C 180,E1 18093.709,E2 18093.709} C_VEL
LIN {X 0,Y 385.896,Z 1176.412,A -85,B 0,C 180,E1 18091.037,E2 18091.037} C_VEL
LIN {X 0,Y 385.831,Z 1177.041,A -85,B 0,C 180,E1 18088.364,E2 18088.364} C_VEL
LIN {X 0,Y 386.049,Z 1175.893,A -85,B 0,C 180,E1 18085.69,E2 18085.69} C_VEL
LIN {X 0,Y 386.553,Z 1173.131,A -85,B 0,C 180,E1 18083.164,E2 18083.164} C_VEL
LIN {X 0,Y 387.396,Z 1168.599,A -85,B 0,C 180,E1 18080.64,E2 18080.64} C_VEL
LIN {X 0,Y 388.632,Z 1162.131,A -85,B 0,C 180,E1 18078.12,E2 18078.12} C_VEL
LIN {X 0,Y 390.217,Z 1154.096,A -85,B 0,C 180,E1 18075.758,E2 18075.758} C_VEL
LIN {X 0,Y 392.088,Z 1144.493,A -85,B 0,C 180,E1 18073.555,E2 18073.555} C_VEL
LIN {X 0,Y 394.163,Z 1133.265,A -85,B 0,C 180,E1 18071.511,E2 18071.511} C_VEL
LIN {X 0,Y 396.277,Z 1120.934,A -85,B 0,C 180,E1 18069.698,E2 18069.698} C_VEL
LIN {X 0,Y 398.333,Z 1107.63,A -85,B 0,C 180,E1 18068.112,E2 18068.112} C_VEL
LIN {X 0,Y 400.206,Z 1093.363,A -85,B 0,C 180,E1 18066.748,E2 18066.748} C_VEL
LIN {X 0,Y 401.84,Z 1078.219,A -85,B 0,C 180,E1 18065.601,E2 18065.601} C_VEL
LIN {X 0,Y 403.199,Z 1061.493,A -85,B 0,C 180,E1 18064.632,E2 18064.632} C_VEL
LIN {X 0,Y 404.101,Z 1044.382,A -85,B 0,C 180,E1 18063.919,E2 18063.919} C_VEL
LIN {X 0,Y 404.48,Z 1025.985,A -85,B 0,C 180,E1 18063.44,E2 18063.44} C_VEL
LIN {X 0,Y 405.161,Z 993.318,A -85,B 0,C 180,E1 18062.85,E2 18062.85} C_VEL
LIN {X 0,Y 404.484,Z 985.706,A -85,B 0,C 180,E1 18062.651,E2 18062.651} C_VEL
LIN {X 0,Y 399.526,Z 965.756,A -85,B 0,C 180,E1 18061.882,E2 18061.882} C_VEL
LIN {X 0,Y 399.086,Z 959.214,A -85,B 0,C 180,E1 18061.717,E2 18061.717} C_VEL
LIN {X 0,Y 401.67,Z 869.364,A -85,B 0,C 180,E1 18060.111,E2 18060.111} C_VEL
LIN {X 0,Y 401.17,Z 864.167,A -85,B 0,C 180,E1 18059.933,E2 18059.933} C_VEL
LIN {X 0,Y 404.775,Z 815.236,A -85,B 0,C 180,E1 18055.976,E2 18055.976} C_VEL
LIN {X 0,Y 409.006,Z 766.964,A -85,B 0,C 180,E1 18051.924,E2 18051.924} C_VEL
LIN {X 0,Y 410.377,Z 753.114,A -85,B 0,C 180,E1 18050.735,E2 18050.735} C_VEL
LIN {X 0,Y 411.914,Z 753.489,A -85,B 0,C 180,E1 18050.505,E2 18050.505} C_VEL
LIN {X 0,Y 414.795,Z 752.167,A -85,B 0,C 180,E1 18050.161,E2 18050.161} C_VEL
LIN {X 0,Y 418.848,Z 748.065,A -85,B 0,C 180,E1 18049.776,E2 18049.776} C_VEL
LIN {X 0,Y 419.751,Z 746.86,A -85,B 0,C 180,E1 18049.702,E2 18049.702} C_VEL
LIN {X 0,Y 423.892,Z 745.035,A -85,B 0,C 180,E1 18049.217,E2 18049.217} C_VEL
LIN {X 0,Y 428.547,Z 740.887,A -85,B 0,C 180,E1 18048.765,E2 18048.765} C_VEL
LIN {X 0,Y 429.835,Z 739.545,A -85,B 0,C 180,E1 18048.649,E2 18048.649} C_VEL
LIN {X 0,Y 434.95,Z 736.567,A -85,B 0,C 180,E1 18048.099,E2 18048.099} C_VEL
LIN {X 0,Y 436.943,Z 735.294,A -85,B 0,C 180,E1 18047.893,E2 18047.893} C_VEL
LIN {X 0,Y 438.527,Z 734.986,A -85,B 0,C 180,E1 18047.706,E2 18047.706} C_VEL
LIN {X 0,Y 445.909,Z 746.592,A -85,B 0,C 180,E1 18046.403,E2 18046.403} C_VEL
LIN {X 0,Y 424.237,Z 977.901,A -85,B 0,C 180,E1 18040.852,E2 18040.852} C_VEL
LIN {X 0,Y 422.078,Z 1001.373,A -85,B 0,C 180,E1 18040.098,E2 18040.098} C_VEL
LIN {X 0,Y 419.435,Z 1022.984,A -85,B 0,C 180,E1 18039.178,E2 18039.178} C_VEL
LIN {X 0,Y 416.079,Z 1045.693,A -85,B 0,C 180,E1 18037.967,E2 18037.967} C_VEL
LIN {X 0,Y 412.462,Z 1066.54,A -85,B 0,C 180,E1 18036.609,E2 18036.609} C_VEL
LIN {X 0,Y 408.351,Z 1087.38,A -85,B 0,C 180,E1 18034.958,E2 18034.958} C_VEL
LIN {X 0,Y 404.016,Z 1107.347,A -85,B 0,C 180,E1 18033.073,E2 18033.073} C_VEL
LIN {X 0,Y 399.739,Z 1125.821,A -85,B 0,C 180,E1 18031.016,E2 18031.016} C_VEL
LIN {X 0,Y 395.449,Z 1143.394,A -85,B 0,C 180,E1 18028.713,E2 18028.713} C_VEL
LIN {X 0,Y 391.42,Z 1159.424,A -85,B 0,C 180,E1 18026.227,E2 18026.227} C_VEL
LIN {X 0,Y 387.546,Z 1174.886,A -85,B 0,C 180,E1 18023.411,E2 18023.411} C_VEL
LIN {X 0,Y 384.343,Z 1188.16,A -85,B 0,C 180,E1 18020.562,E2 18020.562} C_VEL
LIN {X 0,Y 381.599,Z 1200.139,A -85,B 0,C 180,E1 18017.485,E2 18017.485} C_VEL
LIN {X 0,Y 379.496,Z 1210.331,A -85,B 0,C 180,E1 18014.34,E2 18014.34} C_VEL
LIN {X 0,Y 377.97,Z 1219.121,A -85,B 0,C 180,E1 18011.046,E2 18011.046} C_VEL
LIN {X 0,Y 377.062,Z 1225.75,A -85,B 0,C 180,E1 18007.926,E2 18007.926} C_VEL
LIN {X 0,Y 376.522,Z 1231.216,A -85,B 0,C 180,E1 18004.57,E2 18004.57} C_VEL
LIN {X 0,Y 376.326,Z 1234.997,A -85,B 0,C 180,E1 18001.37,E2 18001.37} C_VEL
LIN {X 0,Y 376.29,Z 1237.227,A -85,B 0,C 180,E1 17998.173,E2 17998.173} C_VEL
LIN {X 0,Y 376.377,Z 1238.194,A -85,B 0,C 180,E1 17994.818,E2 17994.818} C_VEL
LIN {X 0,Y 376.629,Z 1237.661,A -85,B 0,C 180,E1 17991.604,E2 17991.604} C_VEL
LIN {X 0,Y 377.166,Z 1235.655,A -85,B 0,C 180,E1 17988.221,E2 17988.221} C_VEL
LIN {X 0,Y 378.234,Z 1232.14,A -85,B 0,C 180,E1 17984.78,E2 17984.78} C_VEL
LIN {X 0,Y 380.011,Z 1226.863,A -85,B 0,C 180,E1 17981.276,E2 17981.276} C_VEL
LIN {X 0,Y 382.561,Z 1220.048,A -85,B 0,C 180,E1 17977.891,E2 17977.891} C_VEL
LIN {X 0,Y 386.037,Z 1211.492,A -85,B 0,C 180,E1 17974.535,E2 17974.535} C_VEL
LIN {X 0,Y 390.307,Z 1201.546,A -85,B 0,C 180,E1 17971.376,E2 17971.376} C_VEL
LIN {X 0,Y 395.247,Z 1190.248,A -85,B 0,C 180,E1 17968.421,E2 17968.421} C_VEL
LIN {X 0,Y 401.385,Z 1176.13,A -85,B 0,C 180,E1 17965.391,E2 17965.391} C_VEL
LIN {X 0,Y 407.787,Z 1161.077,A -85,B 0,C 180,E1 17962.725,E2 17962.725} C_VEL
LIN {X 0,Y 414.603,Z 1144.374,A -85,B 0,C 180,E1 17960.275,E2 17960.275} C_VEL
LIN {X 0,Y 421.277,Z 1127.18,A -85,B 0,C 180,E1 17958.168,E2 17958.168} C_VEL
LIN {X 0,Y 428.112,Z 1108.598,A -85,B 0,C 180,E1 17956.264,E2 17956.264} C_VEL
LIN {X 0,Y 435.908,Z 1086.607,A -85,B 0,C 180,E1 17954.397,E2 17954.397} C_VEL
LIN {X 0,Y 440.176,Z 1074.16,A -85,B 0,C 180,E1 17953.496,E2 17953.496} C_VEL
LIN {X 0,Y 427.442,Z 1097.506,A -85,B 0,C 180,E1 17951.634,E2 17951.634} C_VEL
LIN {X 0,Y 416.565,Z 1119.636,A -85,B 0,C 180,E1 17949.502,E2 17949.502} C_VEL
LIN {X 0,Y 405.826,Z 1145.703,A -85,B 0,C 180,E1 17946.603,E2 17946.603} C_VEL
LIN {X 0,Y 396.748,Z 1172.922,A -85,B 0,C 180,E1 17943.155,E2 17943.155} C_VEL
LIN {X 0,Y 390.086,Z 1197.006,A -85,B 0,C 180,E1 17939.652,E2 17939.652} C_VEL
LIN {X 0,Y 385.601,Z 1215.813,A -85,B 0,C 180,E1 17936.49,E2 17936.49} C_VEL
LIN {X 0,Y 382.306,Z 1231.466,A -85,B 0,C 180,E1 17933.427,E2 17933.427} C_VEL
LIN {X 0,Y 379.862,Z 1244.849,A -85,B 0,C 180,E1 17930.334,E2 17930.334} C_VEL
LIN {X 0,Y 378.113,Z 1255.973,A -85,B 0,C 180,E1 17927.23,E2 17927.23} C_VEL
LIN {X 0,Y 377.041,Z 1264.574,A -85,B 0,C 180,E1 17924.28,E2 17924.28} C_VEL
LIN {X 0,Y 376.44,Z 1271.368,A -85,B 0,C 180,E1 17921.338,E2 17921.338} C_VEL
LIN {X 0,Y 376.202,Z 1276.437,A -85,B 0,C 180,E1 17918.408,E2 17918.408} C_VEL
LIN {X 0,Y 376.182,Z 1279.851,A -85,B 0,C 180,E1 17915.493,E2 17915.493} C_VEL
LIN {X 0,Y 376.255,Z 1281.721,A -85,B 0,C 180,E1 17912.439,E2 17912.439} C_VEL
LIN {X 0,Y 376.309,Z 1281.882,A -85,B 0,C 180,E1 17909.545,E2 17909.545} C_VEL
LIN {X 0,Y 376.29,Z 1280.494,A -85,B 0,C 180,E1 17906.651,E2 17906.651} C_VEL
LIN {X 0,Y 376.25,Z 1277.496,A -85,B 0,C 180,E1 17903.677,E2 17903.677} C_VEL
LIN {X 0,Y 376.315,Z 1272.521,A -85,B 0,C 180,E1 17900.52,E2 17900.52} C_VEL
LIN {X 0,Y 376.665,Z 1265.58,A -85,B 0,C 180,E1 17897.274,E2 17897.274} C_VEL
LIN {X 0,Y 377.432,Z 1256.879,A -85,B 0,C 180,E1 17894.084,E2 17894.084} C_VEL
LIN {X 0,Y 378.826,Z 1245.663,A -85,B 0,C 180,E1 17890.738,E2 17890.738} C_VEL
LIN {X 0,Y 380.795,Z 1233.109,A -85,B 0,C 180,E1 17887.623,E2 17887.623} C_VEL
LIN {X 0,Y 383.492,Z 1218.424,A -85,B 0,C 180,E1 17884.522,E2 17884.522} C_VEL
LIN {X 0,Y 387.2,Z 1200.375,A -85,B 0,C 180,E1 17881.297,E2 17881.297} C_VEL
LIN {X 0,Y 391.414,Z 1181.478,A -85,B 0,C 180,E1 17878.423,E2 17878.423} C_VEL
LIN {X 0,Y 396.029,Z 1161.606,A -85,B 0,C 180,E1 17875.825,E2 17875.825} C_VEL
LIN {X 0,Y 401.133,Z 1140.37,A -85,B 0,C 180,E1 17873.437,E2 17873.437} C_VEL
LIN {X 0,Y 406.629,Z 1117.471,A -85,B 0,C 180,E1 17871.242,E2 17871.242} C_VEL
LIN {X 0,Y 412.791,Z 1091.931,A -85,B 0,C 180,E1 17869.158,E2 17869.158} C_VEL
LIN {X 0,Y 418.389,Z 1068.331,A -85,B 0,C 180,E1 17867.539,E2 17867.539} C_VEL
